LIN {X 0,Y 249.016,Z 307.091,A -85,B 0,C 180,E1 -18932.424,E2 -18932.424} C_VEL
LIN {X 0,Y 249.002,Z 307.055,A -85,B 0,C 180,E1 -18936.346,E2 -18936.346} C_VEL
LIN {X 0,Y 248.968,Z 307.097,A -85,B 0,C 180,E1 -18940.481,E2 -18940.481} C_VEL
LIN {X 0,Y 248.963,Z 307.068,A -85,B 0,C 180,E1 -18944.884,E2 -18944.884} C_VEL
LIN {X 0,Y 248.997,Z 307.08,A -85,B 0,C 180,E1 -18947.359,E2 -18947.359} C_VEL
LIN {X 0,Y 249.012,Z 307.077,A -85,B 0,C 180,E1 -18951.617,E2 -18951.617} C_VEL
LIN {X 0,Y 249.03,Z 307.09,A -85,B 0,C 180,E1 -18955.637,E2 -18955.637} C_VEL
LIN {X 0,Y 249.027,Z 307.069,A -85,B 0,C 180,E1 -18959.47,E2 -18959.47} C_VEL
LIN {X 0,Y 249.054,Z 307.084,A -85,B 0,C 180,E1 -18963.16,E2 -18963.16} C_VEL
LIN {X 0,Y 249.047,Z 307.086,A -85,B 0,C 180,E1 -18966.729,E2 -18966.729} C_VEL
LIN {X 0,Y 249.093,Z 307.073,A -85,B 0,C 180,E1 -18970.21,E2 -18970.21} C_VEL
LIN {X 0,Y 249.188,Z 307.062,A -85,B 0,C 180,E1 -18973.508,E2 -18973.508} C_VEL
LIN {X 0,Y 250.131,Z 309.782,A -85,B 0,C 180,E1 -18973.806,E2 -18973.806} C_VEL
LIN {X 0,Y 252.115,Z 312.374,A -85,B 0,C 180,E1 -18974.302,E2 -18974.302} C_VEL
LIN {X 0,Y 254.328,Z 315.703,A -85,B 0,C 180,E1 -18974.862,E2 -18974.862} C_VEL
LIN {X 0,Y 266.802,Z 335.726,A -85,B 0,C 180,E1 -18977.834,E2 -18977.834} C_VEL
LIN {X 0,Y 270.887,Z 343.151,A -85,B 0,C 180,E1 -18978.761,E2 -18978.761} C_VEL
LIN {X 0,Y 279.656,Z 361.75,A -85,B 0,C 180,E1 -18980.732,E2 -18980.732} C_VEL
LIN {X 0,Y 281.163,Z 365.318,A -85,B 0,C 180,E1 -18981.068,E2 -18981.068} C_VEL
LIN {X 0,Y 277.951,Z 432.372,A -85,B 0,C 180,E1 -18982.814,E2 -18982.814} C_VEL
LIN {X 0,Y 276.086,Z 467.971,A -85,B 0,C 180,E1 -18983.791,E2 -18983.791} C_VEL
LIN {X 0,Y 274.618,Z 483.549,A -85,B 0,C 180,E1 -18984.492,E2 -18984.492} C_VEL
LIN {X 0,Y 272.87,Z 497.522,A -85,B 0,C 180,E1 -18985.383,E2 -18985.383} C_VEL
LIN {X 0,Y 270.76,Z 510.63,A -85,B 0,C 180,E1 -18986.465,E2 -18986.465} C_VEL
LIN {X 0,Y 268.162,Z 524.603,A -85,B 0,C 180,E1 -18987.934,E2 -18987.934} C_VEL
LIN {X 0,Y 265.302,Z 537.524,A -85,B 0,C 180,E1 -18989.62,E2 -18989.62} C_VEL
LIN {X 0,Y 262.375,Z 549.476,A -85,B 0,C 180,E1 -18991.534,E2 -18991.534} C_VEL
LIN {X 0,Y 259.677,Z 559.615,A -85,B 0,C 180,E1 -18993.49,E2 -18993.49} C_VEL
LIN {X 0,Y 256.942,Z 569.913,A -85,B 0,C 180,E1 -18995.887,E2 -18995.887} C_VEL
LIN {X 0,Y 254.456,Z 578.684,A -85,B 0,C 180,E1 -18998.337,E2 -18998.337} C_VEL
LIN {X 0,Y 251.975,Z 587.261,A -85,B 0,C 180,E1 -19001.258,E2 -19001.258} C_VEL
LIN {X 0,Y 250.349,Z 593.389,A -85,B 0,C 180,E1 -19003.804,E2 -19003.804} C_VEL
LIN {X 0,Y 249.079,Z 598.519,A -85,B 0,C 180,E1 -19006.407,E2 -19006.407} C_VEL
LIN {X 0,Y 247.86,Z 603.923,A -85,B 0,C 180,E1 -19009.891,E2 -19009.891} C_VEL
LIN {X 0,Y 247.414,Z 606.081,A -85,B 0,C 180,E1 -19011.67,E2 -19011.67} C_VEL
LIN {X 0,Y 246.878,Z 608.676,A -85,B 0,C 180,E1 -19014.371,E2 -19014.371} C_VEL
LIN {X 0,Y 246.513,Z 610.789,A -85,B 0,C 180,E1 -19017.904,E2 -19017.904} C_VEL
LIN {X 0,Y 246.503,Z 611.519,A -85,B 0,C 180,E1 -19021.211,E2 -19021.211} C_VEL
LIN {X 0,Y 246.752,Z 611.025,A -85,B 0,C 180,E1 -19024.724,E2 -19024.724} C_VEL
LIN {X 0,Y 247.204,Z 609.866,A -85,B 0,C 180,E1 -19027.252,E2 -19027.252} C_VEL
LIN {X 0,Y 248.185,Z 607.218,A -85,B 0,C 180,E1 -19030.638,E2 -19030.638} C_VEL
LIN {X 0,Y 249.435,Z 603.684,A -85,B 0,C 180,E1 -19033.669,E2 -19033.669} C_VEL
LIN {X 0,Y 251.153,Z 599.042,A -85,B 0,C 180,E1 -19036.68,E2 -19036.68} C_VEL
LIN {X 0,Y 253.766,Z 592.279,A -85,B 0,C 180,E1 -19040.061,E2 -19040.061} C_VEL
LIN {X 0,Y 256.692,Z 584.864,A -85,B 0,C 180,E1 -19042.966,E2 -19042.966} C_VEL
LIN {X 0,Y 260.213,Z 575.633,A -85,B 0,C 180,E1 -19045.871,E2 -19045.871} C_VEL
LIN {X 0,Y 263.965,Z 565.524,A -85,B 0,C 180,E1 -19048.426,E2 -19048.426} C_VEL
LIN {X 0,Y 267.881,Z 554.319,A -85,B 0,C 180,E1 -19050.727,E2 -19050.727} C_VEL
LIN {X 0,Y 271.724,Z 542.18,A -85,B 0,C 180,E1 -19052.754,E2 -19052.754} C_VEL
LIN {X 0,Y 275.239,Z 529.729,A -85,B 0,C 180,E1 -19054.442,E2 -19054.442} C_VEL
LIN {X 0,Y 278.7,Z 515.562,A -85,B 0,C 180,E1 -19055.979,E2 -19055.979} C_VEL
LIN {X 0,Y 281.492,Z 501.777,A -85,B 0,C 180,E1 -19057.154,E2 -19057.154} C_VEL
LIN {X 0,Y 283.979,Z 486.513,A -85,B 0,C 180,E1 -19058.136,E2 -19058.136} C_VEL
LIN {X 0,Y 285.813,Z 471.219,A -85,B 0,C 180,E1 -19058.83,E2 -19058.83} C_VEL
LIN {X 0,Y 287.248,Z 451.285,A -85,B 0,C 180,E1 -19059.413,E2 -19059.413} C_VEL
LIN {X 0,Y 292.022,Z 372.427,A -85,B 0,C 180,E1 -19061.462,E2 -19061.462} C_VEL
LIN {X 0,Y 286.413,Z 360.627,A -85,B 0,C 180,E1 -19063.188,E2 -19063.188} C_VEL
LIN {X 0,Y 281.374,Z 351.253,A -85,B 0,C 180,E1 -19064.835,E2 -19064.835} C_VEL
LIN {X 0,Y 279.129,Z 347.273,A -85,B 0,C 180,E1 -19065.603,E2 -19065.603} C_VEL
LIN {X 0,Y 277.373,Z 345.191,A -85,B 0,C 180,E1 -19066.185,E2 -19066.185} C_VEL
LIN {X 0,Y 273.701,Z 343.752,A -85,B 0,C 180,E1 -19067.314,E2 -19067.314} C_VEL
LIN {X 0,Y 270.012,Z 342.607,A -85,B 0,C 180,E1 -19068.512,E2 -19068.512} C_VEL
LIN {X 0,Y 268.191,Z 340.919,A -85,B 0,C 180,E1 -19069.192,E2 -19069.192} C_VEL
LIN {X 0,Y 265.708,Z 337.548,A -85,B 0,C 180,E1 -19070.231,E2 -19070.231} C_VEL
LIN {X 0,Y 263.205,Z 334.014,A -85,B 0,C 180,E1 -19071.359,E2 -19071.359} C_VEL
LIN {X 0,Y 260.47,Z 330.142,A -85,B 0,C 180,E1 -19072.681,E2 -19072.681} C_VEL
LIN {X 0,Y 257.242,Z 326.198,A -85,B 0,C 180,E1 -19074.319,E2 -19074.319} C_VEL
LIN {X 0,Y 256.502,Z 324.959,A -85,B 0,C 180,E1 -19074.746,E2 -19074.746} C_VEL
LIN {X 0,Y 253.726,Z 322.405,A -85,B 0,C 180,E1 -19076.318,E2 -19076.318} C_VEL
LIN {X 0,Y 252.065,Z 319.429,A -85,B 0,C 180,E1 -19077.453,E2 -19077.453} C_VEL
LIN {X 0,Y 249.568,Z 317.316,A -85,B 0,C 180,E1 -19079.095,E2 -19079.095} C_VEL
LIN {X 0,Y 248.14,Z 314.667,A -85,B 0,C 180,E1 -19080.307,E2 -19080.307} C_VEL
LIN {X 0,Y 247.833,Z 313.854,A -85,B 0,C 180,E1 -19080.612,E2 -19080.612} C_VEL
LIN {X 0,Y 244.45,Z 312.125,A -85,B 0,C 180,E1 -19083.505,E2 -19083.505} C_VEL
LIN {X 0,Y 242.871,Z 310.007,A -85,B 0,C 180,E1 -19085.399,E2 -19085.399} C_VEL
LIN {X 0,Y 242.386,Z 308.16,A -85,B 0,C 180,E1 -19086.297,E2 -19086.297} C_VEL
LIN {X 0,Y 242.399,Z 307.915,A -85,B 0,C 180,E1 -19086.662,E2 -19086.662} C_VEL
LIN {X 0,Y 242.255,Z 307.93,A -85,B 0,C 180,E1 -19090.027,E2 -19090.027} C_VEL
LIN {X 0,Y 242.116,Z 307.948,A -85,B 0,C 180,E1 -19095.147,E2 -19095.147} C_VEL
LIN {X 0,Y 242.026,Z 307.964,A -85,B 0,C 180,E1 -19098.63,E2 -19098.63} C_VEL
LIN {X 0,Y 241.976,Z 308.133,A -85,B 0,C 180,E1 -19102.186,E2 -19102.186} C_VEL
LIN {X 0,Y 242.156,Z 308.978,A -85,B 0,C 180,E1 -19103.182,E2 -19103.182} C_VEL
LIN {X 0,Y 243.449,Z 311.446,A -85,B 0,C 180,E1 -19105.09,E2 -19105.09} C_VEL
LIN {X 0,Y 246.087,Z 314.023,A -85,B 0,C 180,E1 -19107.712,E2 -19107.712} C_VEL
LIN {X 0,Y 248.877,Z 317.269,A -85,B 0,C 180,E1 -19110.084,E2 -19110.084} C_VEL
LIN {X 0,Y 252.841,Z 322.416,A -85,B 0,C 180,E1 -19112.839,E2 -19112.839} C_VEL
LIN {X 0,Y 254.527,Z 324.821,A -85,B 0,C 180,E1 -19113.907,E2 -19113.907} C_VEL
LIN {X 0,Y 258.657,Z 330.491,A -85,B 0,C 180,E1 -19116.21,E2 -19116.21} C_VEL
LIN {X 0,Y 262.995,Z 337.089,A -85,B 0,C 180,E1 -19118.372,E2 -19118.372} C_VEL
LIN {X 0,Y 266.544,Z 342.557,A -85,B 0,C 180,E1 -19119.966,E2 -19119.966} C_VEL
LIN {X 0,Y 271.658,Z 351.022,A -85,B 0,C 180,E1 -19122.06,E2 -19122.06} C_VEL
LIN {X 0,Y 277.723,Z 362.338,A -85,B 0,C 180,E1 -19124.337,E2 -19124.337} C_VEL
LIN {X 0,Y 283.163,Z 373.979,A -85,B 0,C 180,E1 -19126.225,E2 -19126.225} C_VEL
LIN {X 0,Y 286.725,Z 382.655,A -85,B 0,C 180,E1 -19127.414,E2 -19127.414} C_VEL
LIN {X 0,Y 281.543,Z 465.569,A -85,B 0,C 180,E1 -19129.593,E2 -19129.593} C_VEL
LIN {X 0,Y 280.06,Z 483.965,A -85,B 0,C 180,E1 -19130.158,E2 -19130.158} C_VEL
LIN {X 0,Y 277.977,Z 499.11,A -85,B 0,C 180,E1 -19130.857,E2 -19130.857} C_VEL
LIN {X 0,Y 275.049,Z 514.438,A -85,B 0,C 180,E1 -19131.829,E2 -19131.829} C_VEL
LIN {X 0,Y 272.261,Z 526.889,A -85,B 0,C 180,E1 -19132.889,E2 -19132.889} C_VEL
LIN {X 0,Y 268.805,Z 540.094,A -85,B 0,C 180,E1 -19134.288,E2 -19134.288} C_VEL
LIN {X 0,Y 265.099,Z 552.623,A -85,B 0,C 180,E1 -19135.943,E2 -19135.943} C_VEL
LIN {X 0,Y 261.071,Z 564.628,A -85,B 0,C 180,E1 -19137.883,E2 -19137.883} C_VEL
LIN {X 0,Y 257.052,Z 575.653,A -85,B 0,C 180,E1 -19140.07,E2 -19140.07} C_VEL
LIN {X 0,Y 253.546,Z 585.071,A -85,B 0,C 180,E1 -19142.366,E2 -19142.366} C_VEL
LIN {X 0,Y 250.098,Z 594.176,A -85,B 0,C 180,E1 -19145.071,E2 -19145.071} C_VEL
LIN {X 0,Y 246.918,Z 601.891,A -85,B 0,C 180,E1 -19147.845,E2 -19147.845} C_VEL
LIN {X 0,Y 244.448,Z 608.314,A -85,B 0,C 180,E1 -19150.694,E2 -19150.694} C_VEL
LIN {X 0,Y 242.358,Z 614.253,A -85,B 0,C 180,E1 -19154.01,E2 -19154.01} C_VEL
LIN {X 0,Y 241.239,Z 617.803,A -85,B 0,C 180,E1 -19156.524,E2 -19156.524} C_VEL
LIN {X 0,Y 240.243,Z 621.431,A -85,B 0,C 180,E1 -19159.892,E2 -19159.892} C_VEL
LIN {X 0,Y 239.787,Z 623.867,A -85,B 0,C 180,E1 -19163.268,E2 -19163.268} C_VEL
LIN {X 0,Y 239.735,Z 625.146,A -85,B 0,C 180,E1 -19166.639,E2 -19166.639} C_VEL
LIN {X 0,Y 239.917,Z 625.227,A -85,B 0,C 180,E1 -19170.001,E2 -19170.001} C_VEL
LIN {X 0,Y 239.763,Z 624.101,A -85,B 0,C 180,E1 -19173.361,E2 -19173.361} C_VEL
LIN {X 0,Y 239.797,Z 621.778,A -85,B 0,C 180,E1 -19176.733,E2 -19176.733} C_VEL
LIN {X 0,Y 240.236,Z 618.206,A -85,B 0,C 180,E1 -19180.11,E2 -19180.11} C_VEL
LIN {X 0,Y 241.096,Z 613.285,A -85,B 0,C 180,E1 -19183.486,E2 -19183.486} C_VEL
LIN {X 0,Y 242.47,Z 606.876,A -85,B 0,C 180,E1 -19186.849,E2 -19186.849} C_VEL
LIN {X 0,Y 244.354,Z 599.957,A -85,B 0,C 180,E1 -19189.752,E2 -19189.752} C_VEL
LIN {X 0,Y 246.748,Z 591.573,A -85,B 0,C 180,E1 -19192.614,E2 -19192.614} C_VEL
LIN {X 0,Y 249.609,Z 581.609,A -85,B 0,C 180,E1 -19195.387,E2 -19195.387} C_VEL
LIN {X 0,Y 252.526,Z 571.082,A -85,B 0,C 180,E1 -19197.786,E2 -19197.786} C_VEL
LIN {X 0,Y 255.946,Z 558.736,A -85,B 0,C 180,E1 -19200.075,E2 -19200.075} C_VEL
LIN {X 0,Y 259.013,Z 546.324,A -85,B 0,C 180,E1 -19201.945,E2 -19201.945} C_VEL
LIN {X 0,Y 261.9,Z 533.658,A -85,B 0,C 180,E1 -19203.485,E2 -19203.485} C_VEL
LIN {X 0,Y 264.741,Z 518.918,A -85,B 0,C 180,E1 -19204.918,E2 -19204.918} C_VEL
LIN {X 0,Y 267.239,Z 503.525,A -85,B 0,C 180,E1 -19206.046,E2 -19206.046} C_VEL
LIN {X 0,Y 269.11,Z 488.092,A -85,B 0,C 180,E1 -19206.859,E2 -19206.859} C_VEL
LIN {X 0,Y 270.398,Z 471.788,A -85,B 0,C 180,E1 -19207.412,E2 -19207.412} C_VEL
LIN {X 0,Y 275.166,Z 376.753,A -85,B 0,C 180,E1 -19209.93,E2 -19209.93} C_VEL
LIN {X 0,Y 266.648,Z 356.753,A -85,B 0,C 180,E1 -19211.945,E2 -19211.945} C_VEL
LIN {X 0,Y 259.613,Z 342.174,A -85,B 0,C 180,E1 -19213.669,E2 -19213.669} C_VEL
LIN {X 0,Y 251.353,Z 326.644,A -85,B 0,C 180,E1 -19215.789,E2 -19215.789} C_VEL
LIN {X 0,Y 244.925,Z 315.683,A -85,B 0,C 180,E1 -19217.526,E2 -19217.526} C_VEL
LIN {X 0,Y 243.366,Z 312.658,A -85,B 0,C 180,E1 -19218.029,E2 -19218.029} C_VEL
LIN {X 0,Y 241.941,Z 307.964,A -85,B 0,C 180,E1 -19220.139,E2 -19220.139} C_VEL
LIN {X 0,Y 241.982,Z 307.956,A -85,B 0,C 180,E1 -19224.411,E2 -19224.411} C_VEL
LIN {X 0,Y 241.951,Z 307.972,A -85,B 0,C 180,E1 -19228.474,E2 -19228.474} C_VEL
LIN {X 0,Y 241.953,Z 307.967,A -85,B 0,C 180,E1 -19232.303,E2 -19232.303} C_VEL
LIN {X 0,Y 241.958,Z 307.969,A -85,B 0,C 180,E1 -19236.003,E2 -19236.003} C_VEL
LIN {X 0,Y 241.986,Z 307.968,A -85,B 0,C 180,E1 -19239.601,E2 -19239.601} C_VEL
LIN {X 0,Y 242.114,Z 307.955,A -85,B 0,C 180,E1 -19243.316,E2 -19243.316} C_VEL
LIN {X 0,Y 242.159,Z 307.905,A -85,B 0,C 180,E1 -19248.276,E2 -19248.276} C_VEL
LIN {X 0,Y 242.356,Z 307.921,A -85,B 0,C 180,E1 -19251.661,E2 -19251.661} C_VEL
LIN {X 0,Y 242.387,Z 307.912,A -85,B 0,C 180,E1 -19253.337,E2 -19253.337} C_VEL
LIN {X 0,Y 242.603,Z 307.858,A -85,B 0,C 180,E1 -19258.337,E2 -19258.337} C_VEL
LIN {X 0,Y 242.612,Z 307.89,A -85,B 0,C 180,E1 -19261.657,E2 -19261.657} C_VEL
LIN {X 0,Y 242.38,Z 307.87,A -85,B 0,C 180,E1 -19266.657,E2 -19266.657} C_VEL
LIN {X 0,Y 242.257,Z 307.924,A -85,B 0,C 180,E1 -19270.021,E2 -19270.021} C_VEL
LIN {X 0,Y 242.128,Z 307.917,A -85,B 0,C 180,E1 -19275.14,E2 -19275.14} C_VEL
LIN {X 0,Y 242.039,Z 307.926,A -85,B 0,C 180,E1 -19278.624,E2 -19278.624} C_VEL
LIN {X 0,Y 241.981,Z 307.967,A -85,B 0,C 180,E1 -19282.18,E2 -19282.18} C_VEL
LIN {X 0,Y 241.978,Z 307.931,A -85,B 0,C 180,E1 -19285.824,E2 -19285.824} C_VEL
LIN {X 0,Y 241.953,Z 307.951,A -85,B 0,C 180,E1 -19289.587,E2 -19289.587} C_VEL
LIN {X 0,Y 241.969,Z 307.962,A -85,B 0,C 180,E1 -19293.49,E2 -19293.49} C_VEL
LIN {X 0,Y 241.972,Z 307.933,A -85,B 0,C 180,E1 -19297.581,E2 -19297.581} C_VEL
LIN {X 0,Y 241.897,Z 307.978,A -85,B 0,C 180,E1 -19301.926,E2 -19301.926} C_VEL
LIN {X 0,Y 241.911,Z 307.952,A -85,B 0,C 180,E1 -19306.572,E2 -19306.572} C_VEL
LIN {X 0,Y 241.944,Z 307.973,A -85,B 0,C 180,E1 -19310.279,E2 -19310.279} C_VEL
LIN {X 0,Y 241.966,Z 307.955,A -85,B 0,C 180,E1 -19314.486,E2 -19314.486} C_VEL
LIN {X 0,Y 241.954,Z 307.955,A -85,B 0,C 180,E1 -19318.477,E2 -19318.477} C_VEL
LIN {X 0,Y 241.987,Z 307.967,A -85,B 0,C 180,E1 -19322.31,E2 -19322.31} C_VEL
LIN {X 0,Y 242.027,Z 307.952,A -85,B 0,C 180,E1 -19326.013,E2 -19326.013} C_VEL
LIN {X 0,Y 242.02,Z 307.951,A -85,B 0,C 180,E1 -19329.606,E2 -19329.606} C_VEL
LIN {X 0,Y 242.078,Z 307.956,A -85,B 0,C 180,E1 -19332.053,E2 -19332.053} C_VEL
LIN {X 0,Y 243.143,Z 310.845,A -85,B 0,C 180,E1 -19332.418,E2 -19332.418} C_VEL
LIN {X 0,Y 245.158,Z 313.379,A -85,B 0,C 180,E1 -19332.948,E2 -19332.948} C_VEL
LIN {X 0,Y 247.321,Z 316.579,A -85,B 0,C 180,E1 -19333.523,E2 -19333.523} C_VEL
LIN {X 0,Y 259.586,Z 335.968,A -85,B 0,C 180,E1 -19336.608,E2 -19336.608} C_VEL
LIN {X 0,Y 265.566,Z 346.45,A -85,B 0,C 180,E1 -19338.019,E2 -19338.019} C_VEL
LIN {X 0,Y 274.158,Z 364.708,A -85,B 0,C 180,E1 -19340.015,E2 -19340.015} C_VEL
LIN {X 0,Y 275.294,Z 367.332,A -85,B 0,C 180,E1 -19340.276,E2 -19340.276} C_VEL
LIN {X 0,Y 272.005,Z 432.87,A -85,B 0,C 180,E1 -19342.009,E2 -19342.009} C_VEL
LIN {X 0,Y 270.137,Z 467.831,A -85,B 0,C 180,E1 -19342.984,E2 -19342.984} C_VEL
LIN {X 0,Y 268.633,Z 483.311,A -85,B 0,C 180,E1 -19343.683,E2 -19343.683} C_VEL
LIN {X 0,Y 266.766,Z 497.727,A -85,B 0,C 180,E1 -19344.614,E2 -19344.614} C_VEL
LIN {X 0,Y 264.417,Z 511.816,A -85,B 0,C 180,E1 -19345.808,E2 -19345.808} C_VEL
LIN {X 0,Y 261.826,Z 525.241,A -85,B 0,C 180,E1 -19347.264,E2 -19347.264} C_VEL
LIN {X 0,Y 258.779,Z 538.408,A -85,B 0,C 180,E1 -19349.027,E2 -19349.027} C_VEL
LIN {X 0,Y 255.508,Z 551.324,A -85,B 0,C 180,E1 -19351.181,E2 -19351.181} C_VEL
LIN {X 0,Y 252.247,Z 563.048,A -85,B 0,C 180,E1 -19353.593,E2 -19353.593} C_VEL
LIN {X 0,Y 249.474,Z 572.876,A -85,B 0,C 180,E1 -19356.063,E2 -19356.063} C_VEL
LIN {X 0,Y 246.611,Z 582.487,A -85,B 0,C 180,E1 -19359.017,E2 -19359.017} C_VEL
LIN {X 0,Y 244.296,Z 590.398,A -85,B 0,C 180,E1 -19362.025,E2 -19362.025} C_VEL
LIN {X 0,Y 242.557,Z 596.906,A -85,B 0,C 180,E1 -19365.115,E2 -19365.115} C_VEL
LIN {X 0,Y 241.081,Z 602.801,A -85,B 0,C 180,E1 -19368.702,E2 -19368.702} C_VEL
LIN {X 0,Y 240.522,Z 605.453,A -85,B 0,C 180,E1 -19370.777,E2 -19370.777} C_VEL
LIN {X 0,Y 239.806,Z 608.805,A -85,B 0,C 180,E1 -19374.222,E2 -19374.222} C_VEL
LIN {X 0,Y 239.417,Z 611.011,A -85,B 0,C 180,E1 -19378.012,E2 -19378.012} C_VEL
LIN {X 0,Y 239.425,Z 611.752,A -85,B 0,C 180,E1 -19381.659,E2 -19381.659} C_VEL
LIN {X 0,Y 239.69,Z 611.275,A -85,B 0,C 180,E1 -19384.822,E2 -19384.822} C_VEL
LIN {X 0,Y 240.238,Z 609.872,A -85,B 0,C 180,E1 -19387.902,E2 -19387.902} C_VEL
LIN {X 0,Y 241.124,Z 607.734,A -85,B 0,C 180,E1 -19390.733,E2 -19390.733} C_VEL
LIN {X 0,Y 242.526,Z 604.064,A -85,B 0,C 180,E1 -19394.063,E2 -19394.063} C_VEL
LIN {X 0,Y 244.357,Z 599.457,A -85,B 0,C 180,E1 -19397.169,E2 -19397.169} C_VEL
LIN {X 0,Y 246.769,Z 593.58,A -85,B 0,C 180,E1 -19400.258,E2 -19400.258} C_VEL
LIN {X 0,Y 249.584,Z 586.808,A -85,B 0,C 180,E1 -19403.103,E2 -19403.103} C_VEL
LIN {X 0,Y 252.832,Z 578.933,A -85,B 0,C 180,E1 -19405.785,E2 -19405.785} C_VEL
LIN {X 0,Y 256.291,Z 570.214,A -85,B 0,C 180,E1 -19408.217,E2 -19408.217} C_VEL
LIN {X 0,Y 260.105,Z 560.007,A -85,B 0,C 180,E1 -19410.566,E2 -19410.566} C_VEL
LIN {X 0,Y 263.927,Z 549.071,A -85,B 0,C 180,E1 -19412.622,E2 -19412.622} C_VEL
LIN {X 0,Y 267.723,Z 537.069,A -85,B 0,C 180,E1 -19414.469,E2 -19414.469} C_VEL
LIN {X 0,Y 271.14,Z 524.776,A -85,B 0,C 180,E1 -19416.016,E2 -19416.016} C_VEL
LIN {X 0,Y 274.554,Z 510.705,A -85,B 0,C 180,E1 -19417.423,E2 -19417.423} C_VEL
LIN {X 0,Y 277.311,Z 496.463,A -85,B 0,C 180,E1 -19418.545,E2 -19418.545} C_VEL
LIN {X 0,Y 279.606,Z 481.581,A -85,B 0,C 180,E1 -19419.41,E2 -19419.41} C_VEL
LIN {X 0,Y 281.278,Z 466.673,A -85,B 0,C 180,E1 -19420.004,E2 -19420.004} C_VEL
LIN {X 0,Y 287.094,Z 375.056,A -85,B 0,C 180,E1 -19422.438,E2 -19422.438} C_VEL
LIN {X 0,Y 281.49,Z 363.189,A -85,B 0,C 180,E1 -19424.281,E2 -19424.281} C_VEL
LIN {X 0,Y 275.852,Z 352.738,A -85,B 0,C 180,E1 -19426.255,E2 -19426.255} C_VEL
LIN {X 0,Y 272.39,Z 346.926,A -85,B 0,C 180,E1 -19427.55,E2 -19427.55} C_VEL
LIN {X 0,Y 268.191,Z 340.919,A -85,B 0,C 180,E1 -19429.192,E2 -19429.192} C_VEL
LIN {X 0,Y 266.423,Z 339.37,A -85,B 0,C 180,E1 -19429.883,E2 -19429.883} C_VEL
LIN {X 0,Y 259.762,Z 338.223,A -85,B 0,C 180,E1 -19432.456,E2 -19432.456} C_VEL
LIN {X 0,Y 258.249,Z 336.615,A -85,B 0,C 180,E1 -19433.186,E2 -19433.186} C_VEL
LIN {X 0,Y 254.764,Z 331.965,A -85,B 0,C 180,E1 -19435.07,E2 -19435.07} C_VEL
LIN {X 0,Y 253,Z 330.233,A -85,B 0,C 180,E1 -19436.081,E2 -19436.081} C_VEL
LIN {X 0,Y 250.763,Z 327.162,A -85,B 0,C 180,E1 -19437.535,E2 -19437.535} C_VEL
LIN {X 0,Y 250.101,Z 326.02,A -85,B 0,C 180,E1 -19438.009,E2 -19438.009} C_VEL
LIN {X 0,Y 247.455,Z 323.32,A -85,B 0,C 180,E1 -19439.901,E2 -19439.901} C_VEL
LIN {X 0,Y 246.027,Z 320.612,A -85,B 0,C 180,E1 -19441.22,E2 -19441.22} C_VEL
LIN {X 0,Y 242.806,Z 318.7,A -85,B 0,C 180,E1 -19444.152,E2 -19444.152} C_VEL
LIN {X 0,Y 241.415,Z 316.36,A -85,B 0,C 180,E1 -19446.06,E2 -19446.06} C_VEL
LIN {X 0,Y 240.961,Z 314.87,A -85,B 0,C 180,E1 -19446.914,E2 -19446.914} C_VEL
LIN {X 0,Y 238.232,Z 313.888,A -85,B 0,C 180,E1 -19453.654,E2 -19453.654} C_VEL
LIN {X 0,Y 238.876,Z 314.332,A -85,B 0,C 180,E1 -19458.885,E2 -19458.885} C_VEL
LIN {X 0,Y 240.472,Z 315.068,A -85,B 0,C 180,E1 -19462.064,E2 -19462.064} C_VEL
LIN {X 0,Y 240.98,Z 316.088,A -85,B 0,C 180,E1 -19462.961,E2 -19462.961} C_VEL
LIN {X 0,Y 242.653,Z 318.901,A -85,B 0,C 180,E1 -19465.349,E2 -19465.349} C_VEL
LIN {X 0,Y 244.671,Z 320.82,A -85,B 0,C 180,E1 -19467.363,E2 -19467.363} C_VEL
LIN {X 0,Y 247.396,Z 324.08,A -85,B 0,C 180,E1 -19469.762,E2 -19469.762} C_VEL
LIN {X 0,Y 250.326,Z 328.216,A -85,B 0,C 180,E1 -19471.929,E2 -19471.929} C_VEL
LIN {X 0,Y 251.962,Z 330.295,A -85,B 0,C 180,E1 -19473.001,E2 -19473.001} C_VEL
LIN {X 0,Y 256.324,Z 336.686,A -85,B 0,C 180,E1 -19475.611,E2 -19475.611} C_VEL
LIN {X 0,Y 260.397,Z 343.002,A -85,B 0,C 180,E1 -19477.724,E2 -19477.724} C_VEL
LIN {X 0,Y 263.994,Z 348.761,A -85,B 0,C 180,E1 -19479.422,E2 -19479.422} C_VEL
LIN {X 0,Y 268.962,Z 357.338,A -85,B 0,C 180,E1 -19481.548,E2 -19481.548} C_VEL
LIN {X 0,Y 274.617,Z 368.304,A -85,B 0,C 180,E1 -19483.765,E2 -19483.765} C_VEL
LIN {X 0,Y 279.332,Z 378.777,A -85,B 0,C 180,E1 -19485.486,E2 -19485.486} C_VEL
LIN {X 0,Y 281.952,Z 385.263,A -85,B 0,C 180,E1 -19486.413,E2 -19486.413} C_VEL
LIN {X 0,Y 275.698,Z 478.622,A -85,B 0,C 180,E1 -19488.915,E2 -19488.915} C_VEL
LIN {X 0,Y 273.701,Z 494.637,A -85,B 0,C 180,E1 -19489.584,E2 -19489.584} C_VEL
LIN {X 0,Y 271.032,Z 509.37,A -85,B 0,C 180,E1 -19490.439,E2 -19490.439} C_VEL
LIN {X 0,Y 267.996,Z 522.795,A -85,B 0,C 180,E1 -19491.479,E2 -19491.479} C_VEL
LIN {X 0,Y 264.329,Z 536.894,A -85,B 0,C 180,E1 -19492.908,E2 -19492.908} C_VEL
LIN {X 0,Y 260.428,Z 549.686,A -85,B 0,C 180,E1 -19494.537,E2 -19494.537} C_VEL
LIN {X 0,Y 256.258,Z 562.072,A -85,B 0,C 180,E1 -19496.502,E2 -19496.502} C_VEL
LIN {X 0,Y 252.28,Z 572.561,A -85,B 0,C 180,E1 -19498.513,E2 -19498.513} C_VEL
LIN {X 0,Y 248.435,Z 582.323,A -85,B 0,C 180,E1 -19500.793,E2 -19500.793} C_VEL
LIN {X 0,Y 244.597,Z 591.931,A -85,B 0,C 180,E1 -19503.555,E2 -19503.555} C_VEL
LIN {X 0,Y 241.139,Z 599.988,A -85,B 0,C 180,E1 -19506.377,E2 -19506.377} C_VEL
LIN {X 0,Y 238.412,Z 606.702,A -85,B 0,C 180,E1 -19509.285,E2 -19509.285} C_VEL
LIN {X 0,Y 235.937,Z 612.924,A -85,B 0,C 180,E1 -19512.671,E2 -19512.671} C_VEL
LIN {X 0,Y 234.272,Z 617.766,A -85,B 0,C 180,E1 -19516.115,E2 -19516.115} C_VEL
LIN {X 0,Y 233.191,Z 621.34,A -85,B 0,C 180,E1 -19519.583,E2 -19519.583} C_VEL
LIN {X 0,Y 232.709,Z 623.721,A -85,B 0,C 180,E1 -19523.062,E2 -19523.062} C_VEL
LIN {X 0,Y 232.644,Z 624.952,A -85,B 0,C 180,E1 -19526.537,E2 -19526.537} C_VEL
LIN {X 0,Y 232.826,Z 625.011,A -85,B 0,C 180,E1 -19530.001,E2 -19530.001} C_VEL
LIN {X 0,Y 232.669,Z 623.839,A -85,B 0,C 180,E1 -19533.464,E2 -19533.464} C_VEL
LIN {X 0,Y 232.736,Z 621.468,A -85,B 0,C 180,E1 -19536.938,E2 -19536.938} C_VEL
LIN {X 0,Y 233.177,Z 617.842,A -85,B 0,C 180,E1 -19540.419,E2 -19540.419} C_VEL
LIN {X 0,Y 234.134,Z 612.866,A -85,B 0,C 180,E1 -19543.895,E2 -19543.895} C_VEL
LIN {X 0,Y 235.593,Z 606.396,A -85,B 0,C 180,E1 -19547.356,E2 -19547.356} C_VEL
LIN {X 0,Y 237.6,Z 599.412,A -85,B 0,C 180,E1 -19550.338,E2 -19550.338} C_VEL
LIN {X 0,Y 240.152,Z 590.971,A -85,B 0,C 180,E1 -19553.271,E2 -19553.271} C_VEL
LIN {X 0,Y 242.996,Z 581.341,A -85,B 0,C 180,E1 -19556.008,E2 -19556.008} C_VEL
LIN {X 0,Y 246.184,Z 570.313,A -85,B 0,C 180,E1 -19558.566,E2 -19558.566} C_VEL
LIN {X 0,Y 249.771,Z 557.816,A -85,B 0,C 180,E1 -19560.898,E2 -19560.898} C_VEL
LIN {X 0,Y 252.951,Z 545.271,A -85,B 0,C 180,E1 -19562.805,E2 -19562.805} C_VEL
LIN {X 0,Y 256.245,Z 531.062,A -85,B 0,C 180,E1 -19564.518,E2 -19564.518} C_VEL
LIN {X 0,Y 259.042,Z 516.269,A -85,B 0,C 180,E1 -19565.923,E2 -19565.923} C_VEL
LIN {X 0,Y 261.504,Z 501.472,A -85,B 0,C 180,E1 -19566.965,E2 -19566.965} C_VEL
LIN {X 0,Y 263.317,Z 486.221,A -85,B 0,C 180,E1 -19567.749,E2 -19567.749} C_VEL
LIN {X 0,Y 264.504,Z 470.602,A -85,B 0,C 180,E1 -19568.274,E2 -19568.274} C_VEL
LIN {X 0,Y 269.295,Z 378.699,A -85,B 0,C 180,E1 -19570.75,E2 -19570.75} C_VEL
LIN {X 0,Y 260.56,Z 358.235,A -85,B 0,C 180,E1 -19572.903,E2 -19572.903} C_VEL
LIN {X 0,Y 252.589,Z 342.055,A -85,B 0,C 180,E1 -19574.944,E2 -19574.944} C_VEL
LIN {X 0,Y 245.867,Z 329.597,A -85,B 0,C 180,E1 -19576.751,E2 -19576.751} C_VEL
LIN {X 0,Y 238.626,Z 317.013,A -85,B 0,C 180,E1 -19578.813,E2 -19578.813} C_VEL
LIN {X 0,Y 235.987,Z 312.514,A -85,B 0,C 180,E1 -19579.626,E2 -19579.626} C_VEL
LIN {X 0,Y 234.929,Z 308.838,A -85,B 0,C 180,E1 -19581.353,E2 -19581.353} C_VEL
LIN {X 0,Y 234.905,Z 308.83,A -85,B 0,C 180,E1 -19585.355,E2 -19585.355} C_VEL
LIN {X 0,Y 234.955,Z 308.838,A -85,B 0,C 180,E1 -19587.421,E2 -19587.421} C_VEL
LIN {X 0,Y 234.894,Z 308.853,A -85,B 0,C 180,E1 -19591.396,E2 -19591.396} C_VEL
LIN {X 0,Y 234.901,Z 308.854,A -85,B 0,C 180,E1 -19595.234,E2 -19595.234} C_VEL
LIN {X 0,Y 234.938,Z 308.852,A -85,B 0,C 180,E1 -19598.96,E2 -19598.96} C_VEL
LIN {X 0,Y 235.056,Z 308.836,A -85,B 0,C 180,E1 -19603.091,E2 -19603.091} C_VEL
LIN {X 0,Y 235.092,Z 308.782,A -85,B 0,C 180,E1 -19607.918,E2 -19607.918} C_VEL
LIN {X 0,Y 235.295,Z 308.798,A -85,B 0,C 180,E1 -19611.408,E2 -19611.408} C_VEL
LIN {X 0,Y 235.338,Z 308.792,A -85,B 0,C 180,E1 -19613.137,E2 -19613.137} C_VEL
LIN {X 0,Y 235.562,Z 308.733,A -85,B 0,C 180,E1 -19618.288,E2 -19618.288} C_VEL
LIN {X 0,Y 235.572,Z 308.767,A -85,B 0,C 180,E1 -19621.707,E2 -19621.707} C_VEL
LIN {X 0,Y 235.331,Z 308.747,A -85,B 0,C 180,E1 -19626.858,E2 -19626.858} C_VEL
LIN {X 0,Y 235.205,Z 308.807,A -85,B 0,C 180,E1 -19630.325,E2 -19630.325} C_VEL
LIN {X 0,Y 235.073,Z 308.788,A -85,B 0,C 180,E1 -19635.606,E2 -19635.606} C_VEL
LIN {X 0,Y 234.979,Z 308.814,A -85,B 0,C 180,E1 -19639.205,E2 -19639.205} C_VEL
LIN {X 0,Y 234.917,Z 308.846,A -85,B 0,C 180,E1 -19642.884,E2 -19642.884} C_VEL
LIN {X 0,Y 234.896,Z 308.805,A -85,B 0,C 180,E1 -19646.663,E2 -19646.663} C_VEL
LIN {X 0,Y 234.885,Z 308.845,A -85,B 0,C 180,E1 -19650.57,E2 -19650.57} C_VEL
LIN {X 0,Y 234.912,Z 308.825,A -85,B 0,C 180,E1 -19654.637,E2 -19654.637} C_VEL
LIN {X 0,Y 234.902,Z 308.831,A -85,B 0,C 180,E1 -19658.933,E2 -19658.933} C_VEL
LIN {X 0,Y 234.846,Z 308.84,A -85,B 0,C 180,E1 -19663.491,E2 -19663.491} C_VEL
LIN {X 0,Y 234.864,Z 308.828,A -85,B 0,C 180,E1 -19666.509,E2 -19666.509} C_VEL
LIN {X 0,Y 234.906,Z 308.84,A -85,B 0,C 180,E1 -19671.076,E2 -19671.076} C_VEL
LIN {X 0,Y 234.912,Z 308.844,A -85,B 0,C 180,E1 -19675.359,E2 -19675.359} C_VEL
LIN {X 0,Y 234.906,Z 308.827,A -85,B 0,C 180,E1 -19679.428,E2 -19679.428} C_VEL
LIN {X 0,Y 234.98,Z 308.83,A -85,B 0,C 180,E1 -19683.792,E2 -19683.792} C_VEL
LIN {X 0,Y 234.983,Z 308.829,A -85,B 0,C 180,E1 -19688.967,E2 -19688.967} C_VEL
LIN {X 0,Y 234.972,Z 308.885,A -85,B 0,C 180,E1 -19690.507,E2 -19690.507} C_VEL
LIN {X 0,Y 236.026,Z 311.746,A -85,B 0,C 180,E1 -19690.88,E2 -19690.88} C_VEL
LIN {X 0,Y 238.141,Z 314.287,A -85,B 0,C 180,E1 -19691.473,E2 -19691.473} C_VEL
LIN {X 0,Y 240.536,Z 317.789,A -85,B 0,C 180,E1 -19692.155,E2 -19692.155} C_VEL
LIN {X 0,Y 248.885,Z 330.678,A -85,B 0,C 180,E1 -19694.41,E2 -19694.41} C_VEL
LIN {X 0,Y 259.076,Z 347.4,A -85,B 0,C 180,E1 -19696.948,E2 -19696.948} C_VEL
LIN {X 0,Y 268.888,Z 368.136,A -85,B 0,C 180,E1 -19699.328,E2 -19699.328} C_VEL
LIN {X 0,Y 269.506,Z 369.78,A -85,B 0,C 180,E1 -19699.482,E2 -19699.482} C_VEL
LIN {X 0,Y 264.27,Z 466.924,A -85,B 0,C 180,E1 -19702.118,E2 -19702.118} C_VEL
LIN {X 0,Y 262.699,Z 482.91,A -85,B 0,C 180,E1 -19702.837,E2 -19702.837} C_VEL
LIN {X 0,Y 260.726,Z 497.8,A -85,B 0,C 180,E1 -19703.81,E2 -19703.81} C_VEL
LIN {X 0,Y 258.451,Z 510.951,A -85,B 0,C 180,E1 -19704.929,E2 -19704.929} C_VEL
LIN {X 0,Y 255.701,Z 524.925,A -85,B 0,C 180,E1 -19706.454,E2 -19706.454} C_VEL
LIN {X 0,Y 252.737,Z 537.411,A -85,B 0,C 180,E1 -19708.137,E2 -19708.137} C_VEL
LIN {X 0,Y 249.489,Z 549.849,A -85,B 0,C 180,E1 -19710.201,E2 -19710.201} C_VEL
LIN {X 0,Y 246.205,Z 561.342,A -85,B 0,C 180,E1 -19712.54,E2 -19712.54} C_VEL
LIN {X 0,Y 243.393,Z 571.102,A -85,B 0,C 180,E1 -19714.969,E2 -19714.969} C_VEL
LIN {X 0,Y 240.508,Z 580.475,A -85,B 0,C 180,E1 -19717.788,E2 -19717.788} C_VEL
LIN {X 0,Y 238.113,Z 588.21,A -85,B 0,C 180,E1 -19720.629,E2 -19720.629} C_VEL
LIN {X 0,Y 236.092,Z 595.16,A -85,B 0,C 180,E1 -19723.776,E2 -19723.776} C_VEL
LIN {X 0,Y 234.718,Z 600.285,A -85,B 0,C 180,E1 -19726.647,E2 -19726.647} C_VEL
LIN {X 0,Y 233.619,Z 605.1,A -85,B 0,C 180,E1 -19730.146,E2 -19730.146} C_VEL
LIN {X 0,Y 232.873,Z 608.1,A -85,B 0,C 180,E1 -19733.099,E2 -19733.099} C_VEL
LIN {X 0,Y 232.569,Z 609.584,A -85,B 0,C 180,E1 -19735.027,E2 -19735.027} C_VEL
LIN {X 0,Y 232.27,Z 611.475,A -85,B 0,C 180,E1 -19738.954,E2 -19738.954} C_VEL
LIN {X 0,Y 232.337,Z 611.945,A -85,B 0,C 180,E1 -19742.123,E2 -19742.123} C_VEL
LIN {X 0,Y 232.656,Z 611.42,A -85,B 0,C 180,E1 -19745.359,E2 -19745.359} C_VEL
LIN {X 0,Y 233.498,Z 609.507,A -85,B 0,C 180,E1 -19749.201,E2 -19749.201} C_VEL
LIN {X 0,Y 234.655,Z 606.815,A -85,B 0,C 180,E1 -19752.364,E2 -19752.364} C_VEL
LIN {X 0,Y 236.223,Z 603.054,A -85,B 0,C 180,E1 -19755.562,E2 -19755.562} C_VEL
LIN {X 0,Y 238.32,Z 598.185,A -85,B 0,C 180,E1 -19758.709,E2 -19758.709} C_VEL
LIN {X 0,Y 241.101,Z 591.823,A -85,B 0,C 180,E1 -19761.907,E2 -19761.907} C_VEL
LIN {X 0,Y 244.406,Z 584.328,A -85,B 0,C 180,E1 -19764.897,E2 -19764.897} C_VEL
LIN {X 0,Y 248.03,Z 575.884,A -85,B 0,C 180,E1 -19767.62,E2 -19767.62} C_VEL
LIN {X 0,Y 252.053,Z 566.022,A -85,B 0,C 180,E1 -19770.207,E2 -19770.207} C_VEL
LIN {X 0,Y 256.385,Z 554.685,A -85,B 0,C 180,E1 -19772.609,E2 -19772.609} C_VEL
LIN {X 0,Y 260.627,Z 542.538,A -85,B 0,C 180,E1 -19774.688,E2 -19774.688} C_VEL
LIN {X 0,Y 264.291,Z 530.592,A -85,B 0,C 180,E1 -19776.358,E2 -19776.358} C_VEL
LIN {X 0,Y 268.092,Z 516.271,A -85,B 0,C 180,E1 -19777.96,E2 -19777.96} C_VEL
LIN {X 0,Y 271.162,Z 502.384,A -85,B 0,C 180,E1 -19779.17,E2 -19779.17} C_VEL
LIN {X 0,Y 273.851,Z 487.187,A -85,B 0,C 180,E1 -19780.169,E2 -19780.169} C_VEL
LIN {X 0,Y 275.877,Z 471.479,A -85,B 0,C 180,E1 -19780.898,E2 -19780.898} C_VEL
LIN {X 0,Y 277.575,Z 448.975,A -85,B 0,C 180,E1 -19781.559,E2 -19781.559} C_VEL
LIN {X 0,Y 282.301,Z 377.818,A -85,B 0,C 180,E1 -19783.449,E2 -19783.449} C_VEL
LIN {X 0,Y 276.87,Z 366.28,A -85,B 0,C 180,E1 -19785.337,E2 -19785.337} C_VEL
LIN {X 0,Y 270.801,Z 354.928,A -85,B 0,C 180,E1 -19787.629,E2 -19787.629} C_VEL
LIN {X 0,Y 265.717,Z 347.206,A -85,B 0,C 180,E1 -19789.689,E2 -19789.689} C_VEL
LIN {X 0,Y 260.792,Z 340.205,A -85,B 0,C 180,E1 -19791.918,E2 -19791.918} C_VEL
LIN {X 0,Y 258.249,Z 336.615,A -85,B 0,C 180,E1 -19793.186,E2 -19793.186} C_VEL
LIN {X 0,Y 256.931,Z 334.75,A -85,B 0,C 180,E1 -19793.882,E2 -19793.882} C_VEL
LIN {X 0,Y 255.43,Z 333.622,A -85,B 0,C 180,E1 -19794.645,E2 -19794.645} C_VEL
LIN {X 0,Y 252.256,Z 332.783,A -85,B 0,C 180,E1 -19796.272,E2 -19796.272} C_VEL
LIN {X 0,Y 249.166,Z 332.487,A -85,B 0,C 180,E1 -19797.997,E2 -19797.997} C_VEL
LIN {X 0,Y 247.165,Z 331.568,A -85,B 0,C 180,E1 -19799.301,E2 -19799.301} C_VEL
LIN {X 0,Y 246.592,Z 330.982,A -85,B 0,C 180,E1 -19799.729,E2 -19799.729} C_VEL
LIN {X 0,Y 244.784,Z 327.86,A -85,B 0,C 180,E1 -19801.366,E2 -19801.366} C_VEL
LIN {X 0,Y 244.478,Z 327.436,A -85,B 0,C 180,E1 -19801.65,E2 -19801.65} C_VEL
LIN {X 0,Y 241.413,Z 325.437,A -85,B 0,C 180,E1 -19804.595,E2 -19804.595} C_VEL
LIN {X 0,Y 240.083,Z 323.076,A -85,B 0,C 180,E1 -19806.542,E2 -19806.542} C_VEL
LIN {X 0,Y 239.645,Z 321.827,A -85,B 0,C 180,E1 -19807.374,E2 -19807.374} C_VEL
LIN {X 0,Y 237.246,Z 320.9,A -85,B 0,C 180,E1 -19813.711,E2 -19813.711} C_VEL
LIN {X 0,Y 237.955,Z 321.401,A -85,B 0,C 180,E1 -19819.076,E2 -19819.076} C_VEL
LIN {X 0,Y 239.374,Z 322.058,A -85,B 0,C 180,E1 -19821.9,E2 -19821.9} C_VEL
LIN {X 0,Y 241.107,Z 325.417,A -85,B 0,C 180,E1 -19824.701,E2 -19824.701} C_VEL
LIN {X 0,Y 243.329,Z 327.682,A -85,B 0,C 180,E1 -19827.073,E2 -19827.073} C_VEL
LIN {X 0,Y 245.711,Z 330.665,A -85,B 0,C 180,E1 -19829.251,E2 -19829.251} C_VEL
LIN {X 0,Y 249.148,Z 335.474,A -85,B 0,C 180,E1 -19831.874,E2 -19831.874} C_VEL
LIN {X 0,Y 254.044,Z 342.859,A -85,B 0,C 180,E1 -19835.004,E2 -19835.004} C_VEL
LIN {X 0,Y 257.704,Z 348.712,A -85,B 0,C 180,E1 -19836.997,E2 -19836.997} C_VEL
LIN {X 0,Y 261.099,Z 354.286,A -85,B 0,C 180,E1 -19838.688,E2 -19838.688} C_VEL
LIN {X 0,Y 265.776,Z 362.669,A -85,B 0,C 180,E1 -19840.804,E2 -19840.804} C_VEL
LIN {X 0,Y 271.097,Z 373.273,A -85,B 0,C 180,E1 -19842.996,E2 -19842.996} C_VEL
LIN {X 0,Y 275.444,Z 383.276,A -85,B 0,C 180,E1 -19844.684,E2 -19844.684} C_VEL
LIN {X 0,Y 277.24,Z 387.736,A -85,B 0,C 180,E1 -19845.349,E2 -19845.349} C_VEL
LIN {X 0,Y 270.98,Z 477.662,A -85,B 0,C 180,E1 -19847.789,E2 -19847.789} C_VEL
LIN {X 0,Y 268.927,Z 493.907,A -85,B 0,C 180,E1 -19848.462,E2 -19848.462} C_VEL
LIN {X 0,Y 266.177,Z 508.701,A -85,B 0,C 180,E1 -19849.322,E2 -19849.322} C_VEL
LIN {X 0,Y 263.018,Z 522.186,A -85,B 0,C 180,E1 -19850.362,E2 -19850.362} C_VEL
LIN {X 0,Y 259.186,Z 536.395,A -85,B 0,C 180,E1 -19851.802,E2 -19851.802} C_VEL
LIN {X 0,Y 255.137,Z 549.218,A -85,B 0,C 180,E1 -19853.44,E2 -19853.44} C_VEL
LIN {X 0,Y 250.784,Z 561.65,A -85,B 0,C 180,E1 -19855.426,E2 -19855.426} C_VEL
LIN {X 0,Y 246.273,Z 573.027,A -85,B 0,C 180,E1 -19857.652,E2 -19857.652} C_VEL
LIN {X 0,Y 242.245,Z 582.649,A -85,B 0,C 180,E1 -19859.971,E2 -19859.971} C_VEL
LIN {X 0,Y 238.228,Z 592.16,A -85,B 0,C 180,E1 -19862.791,E2 -19862.791} C_VEL
LIN {X 0,Y 234.62,Z 600.139,A -85,B 0,C 180,E1 -19865.678,E2 -19865.678} C_VEL
LIN {X 0,Y 231.721,Z 606.806,A -85,B 0,C 180,E1 -19868.658,E2 -19868.658} C_VEL
LIN {X 0,Y 229.097,Z 612.957,A -85,B 0,C 180,E1 -19872.137,E2 -19872.137} C_VEL
LIN {X 0,Y 227.327,Z 617.729,A -85,B 0,C 180,E1 -19875.682,E2 -19875.682} C_VEL
LIN {X 0,Y 226.156,Z 621.25,A -85,B 0,C 180,E1 -19879.255,E2 -19879.255} C_VEL
LIN {X 0,Y 225.622,Z 623.579,A -85,B 0,C 180,E1 -19882.843,E2 -19882.843} C_VEL
LIN {X 0,Y 225.541,Z 624.759,A -85,B 0,C 180,E1 -19886.428,E2 -19886.428} C_VEL
LIN {X 0,Y 225.738,Z 624.788,A -85,B 0,C 180,E1 -19890.001,E2 -19890.001} C_VEL
LIN {X 0,Y 225.578,Z 623.571,A -85,B 0,C 180,E1 -19893.573,E2 -19893.573} C_VEL
LIN {X 0,Y 225.649,Z 621.149,A -85,B 0,C 180,E1 -19897.157,E2 -19897.157} C_VEL
LIN {X 0,Y 226.143,Z 617.467,A -85,B 0,C 180,E1 -19900.747,E2 -19900.747} C_VEL
LIN {X 0,Y 227.185,Z 612.43,A -85,B 0,C 180,E1 -19904.329,E2 -19904.329} C_VEL
LIN {X 0,Y 228.784,Z 605.894,A -85,B 0,C 180,E1 -19907.89,E2 -19907.89} C_VEL
LIN {X 0,Y 230.852,Z 598.828,A -85,B 0,C 180,E1 -19910.96,E2 -19910.96} C_VEL
LIN {X 0,Y 233.576,Z 590.303,A -85,B 0,C 180,E1 -19913.966,E2 -19913.966} C_VEL
LIN {X 0,Y 236.555,Z 580.406,A -85,B 0,C 180,E1 -19916.819,E2 -19916.819} C_VEL
LIN {X 0,Y 239.884,Z 569.43,A -85,B 0,C 180,E1 -19919.389,E2 -19919.389} C_VEL
LIN {X 0,Y 243.308,Z 557.97,A -85,B 0,C 180,E1 -19921.57,E2 -19921.57} C_VEL
LIN {X 0,Y 246.586,Z 545.482,A -85,B 0,C 180,E1 -19923.519,E2 -19923.519} C_VEL
LIN {X 0,Y 249.978,Z 531.388,A -85,B 0,C 180,E1 -19925.265,E2 -19925.265} C_VEL
LIN {X 0,Y 252.86,Z 516.742,A -85,B 0,C 180,E1 -19926.696,E2 -19926.696} C_VEL
LIN {X 0,Y 255.494,Z 501.422,A -85,B 0,C 180,E1 -19927.799,E2 -19927.799} C_VEL
LIN {X 0,Y 257.367,Z 486.252,A -85,B 0,C 180,E1 -19928.594,E2 -19928.594} C_VEL
LIN {X 0,Y 258.59,Z 470.767,A -85,B 0,C 180,E1 -19929.127,E2 -19929.127} C_VEL
LIN {X 0,Y 263.453,Z 380.824,A -85,B 0,C 180,E1 -19931.593,E2 -19931.593} C_VEL
LIN {X 0,Y 255.673,Z 362.32,A -85,B 0,C 180,E1 -19933.6,E2 -19933.6} C_VEL
LIN {X 0,Y 248.364,Z 347.316,A -85,B 0,C 180,E1 -19935.533,E2 -19935.533} C_VEL
LIN {X 0,Y 241.61,Z 334.492,A -85,B 0,C 180,E1 -19937.425,E2 -19937.425} C_VEL
LIN {X 0,Y 234.33,Z 321.814,A -85,B 0,C 180,E1 -19939.563,E2 -19939.563} C_VEL
LIN {X 0,Y 230.623,Z 315.859,A -85,B 0,C 180,E1 -19940.71,E2 -19940.71} C_VEL
LIN {X 0,Y 228.646,Z 312.211,A -85,B 0,C 180,E1 -19941.403,E2 -19941.403} C_VEL
LIN {X 0,Y 227.884,Z 309.731,A -85,B 0,C 180,E1 -19942.691,E2 -19942.691} C_VEL
LIN {X 0,Y 227.88,Z 309.707,A -85,B 0,C 180,E1 -19946.377,E2 -19946.377} C_VEL
LIN {X 0,Y 227.874,Z 309.723,A -85,B 0,C 180,E1 -19950.429,E2 -19950.429} C_VEL
LIN {X 0,Y 227.868,Z 309.731,A -85,B 0,C 180,E1 -19954.416,E2 -19954.416} C_VEL
LIN {X 0,Y 227.92,Z 309.727,A -85,B 0,C 180,E1 -19958.28,E2 -19958.28} C_VEL
LIN {X 0,Y 228.018,Z 309.705,A -85,B 0,C 180,E1 -19963.892,E2 -19963.892} C_VEL
LIN {X 0,Y 228.126,Z 309.664,A -85,B 0,C 180,E1 -19969.345,E2 -19969.345} C_VEL
LIN {X 0,Y 228.29,Z 309.673,A -85,B 0,C 180,E1 -19972.924,E2 -19972.924} C_VEL
LIN {X 0,Y 228.495,Z 309.612,A -85,B 0,C 180,E1 -19978.235,E2 -19978.235} C_VEL
LIN {X 0,Y 228.53,Z 309.643,A -85,B 0,C 180,E1 -19981.759,E2 -19981.759} C_VEL
LIN {X 0,Y 228.268,Z 309.627,A -85,B 0,C 180,E1 -19987.071,E2 -19987.071} C_VEL
LIN {X 0,Y 228.136,Z 309.689,A -85,B 0,C 180,E1 -19990.648,E2 -19990.648} C_VEL
LIN {X 0,Y 228.031,Z 309.684,A -85,B 0,C 180,E1 -19994.271,E2 -19994.271} C_VEL
LIN {X 0,Y 227.931,Z 309.673,A -85,B 0,C 180,E1 -19997.956,E2 -19997.956} C_VEL
LIN {X 0,Y 227.9,Z 309.721,A -85,B 0,C 180,E1 -20002.311,E2 -20002.311} C_VEL
LIN {X 0,Y 227.862,Z 309.681,A -85,B 0,C 180,E1 -20006.562,E2 -20006.562} C_VEL
LIN {X 0,Y 227.86,Z 309.715,A -85,B 0,C 180,E1 -20010.276,E2 -20010.276} C_VEL
LIN {X 0,Y 227.866,Z 309.718,A -85,B 0,C 180,E1 -20013.718,E2 -20013.718} C_VEL
LIN {X 0,Y 227.83,Z 309.698,A -85,B 0,C 180,E1 -20018.089,E2 -20018.089} C_VEL
LIN {X 0,Y 227.776,Z 309.729,A -85,B 0,C 180,E1 -20022.745,E2 -20022.745} C_VEL
LIN {X 0,Y 227.793,Z 309.718,A -85,B 0,C 180,E1 -20027.254,E2 -20027.254} C_VEL
LIN {X 0,Y 227.828,Z 309.71,A -85,B 0,C 180,E1 -20031.906,E2 -20031.906} C_VEL
LIN {X 0,Y 227.866,Z 309.729,A -85,B 0,C 180,E1 -20036.376,E2 -20036.376} C_VEL
LIN {X 0,Y 227.889,Z 309.703,A -85,B 0,C 180,E1 -20040.433,E2 -20040.433} C_VEL
LIN {X 0,Y 227.911,Z 309.705,A -85,B 0,C 180,E1 -20044.424,E2 -20044.424} C_VEL
LIN {X 0,Y 227.941,Z 309.736,A -85,B 0,C 180,E1 -20048.858,E2 -20048.858} C_VEL
LIN {X 0,Y 228.967,Z 312.599,A -85,B 0,C 180,E1 -20049.249,E2 -20049.249} C_VEL
LIN {X 0,Y 231.12,Z 315.219,A -85,B 0,C 180,E1 -20049.893,E2 -20049.893} C_VEL
LIN {X 0,Y 233.266,Z 318.465,A -85,B 0,C 180,E1 -20050.546,E2 -20050.546} C_VEL
LIN {X 0,Y 239.79,Z 328.005,A -85,B 0,C 180,E1 -20052.434,E2 -20052.434} C_VEL
LIN {X 0,Y 251.215,Z 346.411,A -85,B 0,C 180,E1 -20055.489,E2 -20055.489} C_VEL
LIN {X 0,Y 255.927,Z 354.853,A -85,B 0,C 180,E1 -20056.674,E2 -20056.674} C_VEL
LIN {X 0,Y 263.631,Z 371.644,A -85,B 0,C 180,E1 -20058.615,E2 -20058.615} C_VEL
LIN {X 0,Y 258.396,Z 466.721,A -85,B 0,C 180,E1 -20061.248,E2 -20061.248} C_VEL
LIN {X 0,Y 256.863,Z 482.149,A -85,B 0,C 180,E1 -20061.939,E2 -20061.939} C_VEL
LIN {X 0,Y 254.707,Z 497.9,A -85,B 0,C 180,E1 -20062.973,E2 -20062.973} C_VEL
LIN {X 0,Y 252.212,Z 511.975,A -85,B 0,C 180,E1 -20064.202,E2 -20064.202} C_VEL
LIN {X 0,Y 249.359,Z 525.802,A -85,B 0,C 180,E1 -20065.757,E2 -20065.757} C_VEL
LIN {X 0,Y 246.191,Z 538.588,A -85,B 0,C 180,E1 -20067.535,E2 -20067.535} C_VEL
LIN {X 0,Y 242.616,Z 551.64,A -85,B 0,C 180,E1 -20069.792,E2 -20069.792} C_VEL
LIN {X 0,Y 239.132,Z 563.399,A -85,B 0,C 180,E1 -20072.321,E2 -20072.321} C_VEL
LIN {X 0,Y 235.885,Z 573.961,A -85,B 0,C 180,E1 -20075.127,E2 -20075.127} C_VEL
LIN {X 0,Y 233.182,Z 582.433,A -85,B 0,C 180,E1 -20077.867,E2 -20077.867} C_VEL
LIN {X 0,Y 230.446,Z 591,A -85,B 0,C 180,E1 -20081.294,E2 -20081.294} C_VEL
LIN {X 0,Y 228.736,Z 596.858,A -85,B 0,C 180,E1 -20084.228,E2 -20084.228} C_VEL
LIN {X 0,Y 227.102,Z 602.855,A -85,B 0,C 180,E1 -20088.026,E2 -20088.026} C_VEL
LIN {X 0,Y 226.188,Z 606.639,A -85,B 0,C 180,E1 -20091.239,E2 -20091.239} C_VEL
LIN {X 0,Y 225.624,Z 609.017,A -85,B 0,C 180,E1 -20093.886,E2 -20093.886} C_VEL
LIN {X 0,Y 225.212,Z 611.326,A -85,B 0,C 180,E1 -20097.909,E2 -20097.909} C_VEL
LIN {X 0,Y 225.151,Z 611.936,A -85,B 0,C 180,E1 -20099.961,E2 -20099.961} C_VEL
LIN {X 0,Y 225.272,Z 612.132,A -85,B 0,C 180,E1 -20102.619,E2 -20102.619} C_VEL
LIN {X 0,Y 225.689,Z 611.439,A -85,B 0,C 180,E1 -20106.273,E2 -20106.273} C_VEL
LIN {X 0,Y 226.366,Z 610.044,A -85,B 0,C 180,E1 -20109.094,E2 -20109.094} C_VEL
LIN {X 0,Y 227.712,Z 607.153,A -85,B 0,C 180,E1 -20112.763,E2 -20112.763} C_VEL
LIN {X 0,Y 229.379,Z 603.456,A -85,B 0,C 180,E1 -20116.053,E2 -20116.053} C_VEL
LIN {X 0,Y 231.653,Z 598.565,A -85,B 0,C 180,E1 -20119.326,E2 -20119.326} C_VEL
LIN {X 0,Y 234.89,Z 591.654,A -85,B 0,C 180,E1 -20122.886,E2 -20122.886} C_VEL
LIN {X 0,Y 238.408,Z 584.063,A -85,B 0,C 180,E1 -20125.942,E2 -20125.942} C_VEL
LIN {X 0,Y 242.787,Z 574.375,A -85,B 0,C 180,E1 -20129.055,E2 -20129.055} C_VEL
LIN {X 0,Y 247.265,Z 563.774,A -85,B 0,C 180,E1 -20131.773,E2 -20131.773} C_VEL
LIN {X 0,Y 251.845,Z 552.151,A -85,B 0,C 180,E1 -20134.15,E2 -20134.15} C_VEL
LIN {X 0,Y 256.088,Z 540.114,A -85,B 0,C 180,E1 -20136.144,E2 -20136.144} C_VEL
LIN {X 0,Y 259.823,Z 528.133,A -85,B 0,C 180,E1 -20137.751,E2 -20137.751} C_VEL
LIN {X 0,Y 263.603,Z 514.152,A -85,B 0,C 180,E1 -20139.252,E2 -20139.252} C_VEL
LIN {X 0,Y 266.615,Z 500.579,A -85,B 0,C 180,E1 -20140.4,E2 -20140.4} C_VEL
LIN {X 0,Y 269.237,Z 485.763,A -85,B 0,C 180,E1 -20141.351,E2 -20141.351} C_VEL
LIN {X 0,Y 271.205,Z 470.78,A -85,B 0,C 180,E1 -20142.024,E2 -20142.024} C_VEL
LIN {X 0,Y 273.143,Z 445.109,A -85,B 0,C 180,E1 -20142.772,E2 -20142.772} C_VEL
LIN {X 0,Y 277.596,Z 380.511,A -85,B 0,C 180,E1 -20144.507,E2 -20144.507} C_VEL
LIN {X 0,Y 272.171,Z 368.888,A -85,B 0,C 180,E1 -20146.533,E2 -20146.533} C_VEL
LIN {X 0,Y 267.092,Z 359.411,A -85,B 0,C 180,E1 -20148.563,E2 -20148.563} C_VEL
LIN {X 0,Y 261.518,Z 350.837,A -85,B 0,C 180,E1 -20150.986,E2 -20150.986} C_VEL
LIN {X 0,Y 257.721,Z 345.541,A -85,B 0,C 180,E1 -20152.826,E2 -20152.826} C_VEL
LIN {X 0,Y 255.065,Z 341.685,A -85,B 0,C 180,E1 -20154.231,E2 -20154.231} C_VEL
LIN {X 0,Y 252.065,Z 337.664,A -85,B 0,C 180,E1 -20155.984,E2 -20155.984} C_VEL
LIN {X 0,Y 249.355,Z 334.479,A -85,B 0,C 180,E1 -20157.714,E2 -20157.714} C_VEL
LIN {X 0,Y 248.162,Z 332.524,A -85,B 0,C 180,E1 -20158.583,E2 -20158.583} C_VEL
LIN {X 0,Y 246.592,Z 330.982,A -85,B 0,C 180,E1 -20159.729,E2 -20159.729} C_VEL
LIN {X 0,Y 245.443,Z 330.398,A -85,B 0,C 180,E1 -20160.597,E2 -20160.597} C_VEL
LIN {X 0,Y 243.365,Z 331.459,A -85,B 0,C 180,E1 -20162.072,E2 -20162.072} C_VEL
LIN {X 0,Y 241.407,Z 332.803,A -85,B 0,C 180,E1 -20163.584,E2 -20163.584} C_VEL
LIN {X 0,Y 240.47,Z 332.623,A -85,B 0,C 180,E1 -20164.515,E2 -20164.515} C_VEL
LIN {X 0,Y 238.856,Z 330.009,A -85,B 0,C 180,E1 -20166.868,E2 -20166.868} C_VEL
LIN {X 0,Y 238.486,Z 328.815,A -85,B 0,C 180,E1 -20167.623,E2 -20167.623} C_VEL
LIN {X 0,Y 236.264,Z 327.93,A -85,B 0,C 180,E1 -20173.769,E2 -20173.769} C_VEL
LIN {X 0,Y 236.961,Z 328.429,A -85,B 0,C 180,E1 -20179.044,E2 -20179.044} C_VEL
LIN {X 0,Y 238.279,Z 329.05,A -85,B 0,C 180,E1 -20181.736,E2 -20181.736} C_VEL
LIN {X 0,Y 239.441,Z 331.67,A -85,B 0,C 180,E1 -20183.805,E2 -20183.805} C_VEL
LIN {X 0,Y 241.998,Z 334.593,A -85,B 0,C 180,E1 -20186.789,E2 -20186.789} C_VEL
LIN {X 0,Y 243.966,Z 337.051,A -85,B 0,C 180,E1 -20188.65,E2 -20188.65} C_VEL
LIN {X 0,Y 247.382,Z 342.06,A -85,B 0,C 180,E1 -20191.418,E2 -20191.418} C_VEL
LIN {X 0,Y 251.756,Z 348.906,A -85,B 0,C 180,E1 -20194.338,E2 -20194.338} C_VEL
LIN {X 0,Y 255.841,Z 355.721,A -85,B 0,C 180,E1 -20196.673,E2 -20196.673} C_VEL
LIN {X 0,Y 258.668,Z 360.584,A -85,B 0,C 180,E1 -20198.134,E2 -20198.134} C_VEL
LIN {X 0,Y 263.048,Z 368.745,A -85,B 0,C 180,E1 -20200.211,E2 -20200.211} C_VEL
LIN {X 0,Y 267.694,Z 378.419,A -85,B 0,C 180,E1 -20202.236,E2 -20202.236} C_VEL
LIN {X 0,Y 271.684,Z 387.877,A -85,B 0,C 180,E1 -20203.871,E2 -20203.871} C_VEL
LIN {X 0,Y 272.669,Z 390.799,A -85,B 0,C 180,E1 -20204.286,E2 -20204.286} C_VEL
LIN {X 0,Y 266.261,Z 478.223,A -85,B 0,C 180,E1 -20206.666,E2 -20206.666} C_VEL
LIN {X 0,Y 264.124,Z 494.147,A -85,B 0,C 180,E1 -20207.339,E2 -20207.339} C_VEL
LIN {X 0,Y 261.165,Z 509.383,A -85,B 0,C 180,E1 -20208.241,E2 -20208.241} C_VEL
LIN {X 0,Y 257.662,Z 523.614,A -85,B 0,C 180,E1 -20209.369,E2 -20209.369} C_VEL
LIN {X 0,Y 253.703,Z 537.455,A -85,B 0,C 180,E1 -20210.82,E2 -20210.82} C_VEL
LIN {X 0,Y 249.093,Z 551.221,A -85,B 0,C 180,E1 -20212.657,E2 -20212.657} C_VEL
LIN {X 0,Y 244.997,Z 562.288,A -85,B 0,C 180,E1 -20214.488,E2 -20214.488} C_VEL
LIN {X 0,Y 240.329,Z 573.528,A -85,B 0,C 180,E1 -20216.75,E2 -20216.75} C_VEL
LIN {X 0,Y 236.128,Z 583.035,A -85,B 0,C 180,E1 -20219.11,E2 -20219.11} C_VEL
LIN {X 0,Y 231.904,Z 592.425,A -85,B 0,C 180,E1 -20221.984,E2 -20221.984} C_VEL
LIN {X 0,Y 228.148,Z 600.295,A -85,B 0,C 180,E1 -20224.942,E2 -20224.942} C_VEL
LIN {X 0,Y 225.069,Z 606.89,A -85,B 0,C 180,E1 -20227.995,E2 -20227.995} C_VEL
LIN {X 0,Y 222.269,Z 612.992,A -85,B 0,C 180,E1 -20231.568,E2 -20231.568} C_VEL
LIN {X 0,Y 220.403,Z 617.714,A -85,B 0,C 180,E1 -20235.222,E2 -20235.222} C_VEL
LIN {X 0,Y 219.14,Z 621.166,A -85,B 0,C 180,E1 -20238.907,E2 -20238.907} C_VEL
LIN {X 0,Y 218.558,Z 623.438,A -85,B 0,C 180,E1 -20242.611,E2 -20242.611} C_VEL
LIN {X 0,Y 218.456,Z 624.566,A -85,B 0,C 180,E1 -20246.312,E2 -20246.312} C_VEL
LIN {X 0,Y 218.651,Z 624.551,A -85,B 0,C 180,E1 -20250.001,E2 -20250.001} C_VEL
LIN {X 0,Y 218.485,Z 623.3,A -85,B 0,C 180,E1 -20253.689,E2 -20253.689} C_VEL
LIN {X 0,Y 218.582,Z 620.822,A -85,B 0,C 180,E1 -20257.39,E2 -20257.39} C_VEL
LIN {X 0,Y 219.122,Z 617.082,A -85,B 0,C 180,E1 -20261.096,E2 -20261.096} C_VEL
LIN {X 0,Y 220.229,Z 611.98,A -85,B 0,C 180,E1 -20264.792,E2 -20264.792} C_VEL
LIN {X 0,Y 221.959,Z 605.375,A -85,B 0,C 180,E1 -20268.46,E2 -20268.46} C_VEL
LIN {X 0,Y 224.133,Z 598.233,A -85,B 0,C 180,E1 -20271.619,E2 -20271.619} C_VEL
LIN {X 0,Y 227.018,Z 589.624,A -85,B 0,C 180,E1 -20274.704,E2 -20274.704} C_VEL
LIN {X 0,Y 229.771,Z 580.856,A -85,B 0,C 180,E1 -20277.31,E2 -20277.31} C_VEL
LIN {X 0,Y 233.03,Z 570.467,A -85,B 0,C 180,E1 -20279.843,E2 -20279.843} C_VEL
LIN {X 0,Y 236.861,Z 558.108,A -85,B 0,C 180,E1 -20282.282,E2 -20282.282} C_VEL
LIN {X 0,Y 240.614,Z 544.293,A -85,B 0,C 180,E1 -20284.466,E2 -20284.466} C_VEL
LIN {X 0,Y 243.785,Z 531.6,A -85,B 0,C 180,E1 -20286.06,E2 -20286.06} C_VEL
LIN {X 0,Y 246.726,Z 517.2,A -85,B 0,C 180,E1 -20287.507,E2 -20287.507} C_VEL
LIN {X 0,Y 249.306,Z 502.807,A -85,B 0,C 180,E1 -20288.587,E2 -20288.587} C_VEL
LIN {X 0,Y 251.367,Z 487.341,A -85,B 0,C 180,E1 -20289.434,E2 -20289.434} C_VEL
LIN {X 0,Y 252.647,Z 472.529,A -85,B 0,C 180,E1 -20289.972,E2 -20289.972} C_VEL
LIN {X 0,Y 257.637,Z 382.677,A -85,B 0,C 180,E1 -20292.489,E2 -20292.489} C_VEL
LIN {X 0,Y 249.799,Z 364.197,A -85,B 0,C 180,E1 -20294.587,E2 -20294.587} C_VEL
LIN {X 0,Y 241.793,Z 347.729,A -85,B 0,C 180,E1 -20296.827,E2 -20296.827} C_VEL
LIN {X 0,Y 233.991,Z 333.398,A -85,B 0,C 180,E1 -20299.12,E2 -20299.12} C_VEL
LIN {X 0,Y 227.017,Z 321.467,A -85,B 0,C 180,E1 -20301.335,E2 -20301.335} C_VEL
LIN {X 0,Y 223.588,Z 316.003,A -85,B 0,C 180,E1 -20302.482,E2 -20302.482} C_VEL
LIN {X 0,Y 221.147,Z 311.95,A -85,B 0,C 180,E1 -20303.352,E2 -20303.352} C_VEL
LIN {X 0,Y 220.826,Z 310.593,A -85,B 0,C 180,E1 -20304.067,E2 -20304.067} C_VEL
LIN {X 0,Y 220.813,Z 310.596,A -85,B 0,C 180,E1 -20307.24,E2 -20307.24} C_VEL
LIN {X 0,Y 220.795,Z 310.61,A -85,B 0,C 180,E1 -20311.478,E2 -20311.478} C_VEL
LIN {X 0,Y 220.798,Z 310.607,A -85,B 0,C 180,E1 -20315.554,E2 -20315.554} C_VEL
LIN {X 0,Y 220.849,Z 310.601,A -85,B 0,C 180,E1 -20319.507,E2 -20319.507} C_VEL
LIN {X 0,Y 220.977,Z 310.587,A -85,B 0,C 180,E1 -20323.364,E2 -20323.364} C_VEL
LIN {X 0,Y 221.052,Z 310.539,A -85,B 0,C 180,E1 -20329,E2 -20329} C_VEL
LIN {X 0,Y 221.228,Z 310.552,A -85,B 0,C 180,E1 -20332.697,E2 -20332.697} C_VEL
LIN {X 0,Y 221.432,Z 310.49,A -85,B 0,C 180,E1 -20338.178,E2 -20338.178} C_VEL
LIN {X 0,Y 221.537,Z 310.504,A -85,B 0,C 180,E1 -20339.997,E2 -20339.997} C_VEL
LIN {X 0,Y 221.463,Z 310.523,A -85,B 0,C 180,E1 -20341.816,E2 -20341.816} C_VEL
LIN {X 0,Y 221.209,Z 310.507,A -85,B 0,C 180,E1 -20347.298,E2 -20347.298} C_VEL
LIN {X 0,Y 221.057,Z 310.572,A -85,B 0,C 180,E1 -20350.994,E2 -20350.994} C_VEL
LIN {X 0,Y 220.973,Z 310.534,A -85,B 0,C 180,E1 -20356.63,E2 -20356.63} C_VEL
LIN {X 0,Y 220.862,Z 310.589,A -85,B 0,C 180,E1 -20360.485,E2 -20360.485} C_VEL
LIN {X 0,Y 220.797,Z 310.586,A -85,B 0,C 180,E1 -20364.439,E2 -20364.439} C_VEL
LIN {X 0,Y 220.783,Z 310.569,A -85,B 0,C 180,E1 -20368.517,E2 -20368.517} C_VEL
LIN {X 0,Y 220.802,Z 310.605,A -85,B 0,C 180,E1 -20372.754,E2 -20372.754} C_VEL
LIN {X 0,Y 220.791,Z 310.566,A -85,B 0,C 180,E1 -20377.272,E2 -20377.272} C_VEL
LIN {X 0,Y 220.738,Z 310.614,A -85,B 0,C 180,E1 -20381.955,E2 -20381.955} C_VEL
LIN {X 0,Y 220.751,Z 310.579,A -85,B 0,C 180,E1 -20385.54,E2 -20385.54} C_VEL
LIN {X 0,Y 220.794,Z 310.604,A -85,B 0,C 180,E1 -20390.461,E2 -20390.461} C_VEL
LIN {X 0,Y 220.813,Z 310.578,A -85,B 0,C 180,E1 -20392.791,E2 -20392.791} C_VEL
LIN {X 0,Y 220.802,Z 310.605,A -85,B 0,C 180,E1 -20397.241,E2 -20397.241} C_VEL
LIN {X 0,Y 220.813,Z 310.596,A -85,B 0,C 180,E1 -20401.483,E2 -20401.483} C_VEL
LIN {X 0,Y 220.848,Z 310.585,A -85,B 0,C 180,E1 -20405.563,E2 -20405.563} C_VEL
LIN {X 0,Y 220.859,Z 310.707,A -85,B 0,C 180,E1 -20407.05,E2 -20407.05} C_VEL
LIN {X 0,Y 221.858,Z 313.435,A -85,B 0,C 180,E1 -20407.458,E2 -20407.458} C_VEL
LIN {X 0,Y 224.208,Z 316.191,A -85,B 0,C 180,E1 -20408.217,E2 -20408.217} C_VEL
LIN {X 0,Y 226.521,Z 319.626,A -85,B 0,C 180,E1 -20408.975,E2 -20408.975} C_VEL
LIN {X 0,Y 235.392,Z 332.592,A -85,B 0,C 180,E1 -20411.671,E2 -20411.671} C_VEL
LIN {X 0,Y 247.244,Z 351.934,A -85,B 0,C 180,E1 -20414.953,E2 -20414.953} C_VEL
LIN {X 0,Y 251.217,Z 359.356,A -85,B 0,C 180,E1 -20416,E2 -20416} C_VEL
LIN {X 0,Y 257.92,Z 373.938,A -85,B 0,C 180,E1 -20417.742,E2 -20417.742} C_VEL
LIN {X 0,Y 252.471,Z 467.789,A -85,B 0,C 180,E1 -20420.385,E2 -20420.385} C_VEL
LIN {X 0,Y 250.77,Z 483.73,A -85,B 0,C 180,E1 -20421.133,E2 -20421.133} C_VEL
LIN {X 0,Y 248.657,Z 498.53,A -85,B 0,C 180,E1 -20422.14,E2 -20422.14} C_VEL
LIN {X 0,Y 245.988,Z 512.96,A -85,B 0,C 180,E1 -20423.437,E2 -20423.437} C_VEL
LIN {X 0,Y 243.046,Z 526.643,A -85,B 0,C 180,E1 -20425.023,E2 -20425.023} C_VEL
LIN {X 0,Y 239.557,Z 540.116,A -85,B 0,C 180,E1 -20426.965,E2 -20426.965} C_VEL
LIN {X 0,Y 236.091,Z 552.277,A -85,B 0,C 180,E1 -20429.147,E2 -20429.147} C_VEL
LIN {X 0,Y 232.485,Z 563.947,A -85,B 0,C 180,E1 -20431.732,E2 -20431.732} C_VEL
LIN {X 0,Y 229.373,Z 573.749,A -85,B 0,C 180,E1 -20434.392,E2 -20434.392} C_VEL
LIN {X 0,Y 226.18,Z 583.313,A -85,B 0,C 180,E1 -20437.588,E2 -20437.588} C_VEL
LIN {X 0,Y 223.57,Z 591.227,A -85,B 0,C 180,E1 -20440.871,E2 -20440.871} C_VEL
LIN {X 0,Y 221.829,Z 596.82,A -85,B 0,C 180,E1 -20443.745,E2 -20443.745} C_VEL
LIN {X 0,Y 220.1,Z 602.919,A -85,B 0,C 180,E1 -20447.693,E2 -20447.693} C_VEL
LIN {X 0,Y 219.231,Z 606.386,A -85,B 0,C 180,E1 -20450.647,E2 -20450.647} C_VEL
LIN {X 0,Y 218.41,Z 609.818,A -85,B 0,C 180,E1 -20454.727,E2 -20454.727} C_VEL
LIN {X 0,Y 218.183,Z 610.995,A -85,B 0,C 180,E1 -20456.804,E2 -20456.804} C_VEL
LIN {X 0,Y 218.054,Z 611.981,A -85,B 0,C 180,E1 -20459.523,E2 -20459.523} C_VEL
LIN {X 0,Y 218.223,Z 612.318,A -85,B 0,C 180,E1 -20463.194,E2 -20463.194} C_VEL
LIN {X 0,Y 218.639,Z 611.69,A -85,B 0,C 180,E1 -20466.53,E2 -20466.53} C_VEL
LIN {X 0,Y 219.47,Z 610.095,A -85,B 0,C 180,E1 -20469.823,E2 -20469.823} C_VEL
LIN {X 0,Y 220.653,Z 607.78,A -85,B 0,C 180,E1 -20472.903,E2 -20472.903} C_VEL
LIN {X 0,Y 222.559,Z 603.871,A -85,B 0,C 180,E1 -20476.575,E2 -20476.575} C_VEL
LIN {X 0,Y 224.967,Z 599.012,A -85,B 0,C 180,E1 -20479.938,E2 -20479.938} C_VEL
LIN {X 0,Y 228.653,Z 591.699,A -85,B 0,C 180,E1 -20483.81,E2 -20483.81} C_VEL
LIN {X 0,Y 232.507,Z 583.823,A -85,B 0,C 180,E1 -20487.042,E2 -20487.042} C_VEL
LIN {X 0,Y 237.048,Z 574.291,A -85,B 0,C 180,E1 -20490.132,E2 -20490.132} C_VEL
LIN {X 0,Y 241.578,Z 564.062,A -85,B 0,C 180,E1 -20492.789,E2 -20492.789} C_VEL
LIN {X 0,Y 246.371,Z 552.376,A -85,B 0,C 180,E1 -20495.215,E2 -20495.215} C_VEL
LIN {X 0,Y 251.205,Z 539.173,A -85,B 0,C 180,E1 -20497.4,E2 -20497.4} C_VEL
LIN {X 0,Y 255.148,Z 527.022,A -85,B 0,C 180,E1 -20499.021,E2 -20499.021} C_VEL
LIN {X 0,Y 259.043,Z 512.878,A -85,B 0,C 180,E1 -20500.52,E2 -20500.52} C_VEL
LIN {X 0,Y 262.341,Z 498.015,A -85,B 0,C 180,E1 -20501.742,E2 -20501.742} C_VEL
LIN {X 0,Y 265.039,Z 482.598,A -85,B 0,C 180,E1 -20502.664,E2 -20502.664} C_VEL
LIN {X 0,Y 266.874,Z 468.107,A -85,B 0,C 180,E1 -20503.265,E2 -20503.265} C_VEL
LIN {X 0,Y 273.007,Z 383.244,A -85,B 0,C 180,E1 -20505.604,E2 -20505.604} C_VEL
LIN {X 0,Y 267.895,Z 372.276,A -85,B 0,C 180,E1 -20507.64,E2 -20507.64} C_VEL
LIN {X 0,Y 263.593,Z 364.08,A -85,B 0,C 180,E1 -20509.487,E2 -20509.487} C_VEL
LIN {X 0,Y 258.502,Z 356.176,A -85,B 0,C 180,E1 -20511.83,E2 -20511.83} C_VEL
LIN {X 0,Y 254.898,Z 351,A -85,B 0,C 180,E1 -20513.671,E2 -20513.671} C_VEL
LIN {X 0,Y 252.726,Z 347.79,A -85,B 0,C 180,E1 -20514.896,E2 -20514.896} C_VEL
LIN {X 0,Y 250.186,Z 344.212,A -85,B 0,C 180,E1 -20516.453,E2 -20516.453} C_VEL
LIN {X 0,Y 247.433,Z 340.87,A -85,B 0,C 180,E1 -20518.278,E2 -20518.278} C_VEL
LIN {X 0,Y 246.259,Z 338.983,A -85,B 0,C 180,E1 -20519.185,E2 -20519.185} C_VEL
LIN {X 0,Y 243.713,Z 335.653,A -85,B 0,C 180,E1 -20521.321,E2 -20521.321} C_VEL
LIN {X 0,Y 242.954,Z 334.278,A -85,B 0,C 180,E1 -20522.075,E2 -20522.075} C_VEL
LIN {X 0,Y 240.47,Z 332.623,A -85,B 0,C 180,E1 -20524.515,E2 -20524.515} C_VEL
LIN {X 0,Y 239.323,Z 332.075,A -85,B 0,C 180,E1 -20525.898,E2 -20525.898} C_VEL
LIN {X 0,Y 237.497,Z 333.141,A -85,B 0,C 180,E1 -20528.234,E2 -20528.234} C_VEL
LIN {X 0,Y 235.878,Z 334.987,A -85,B 0,C 180,E1 -20531.099,E2 -20531.099} C_VEL
LIN {X 0,Y 235.577,Z 335.118,A -85,B 0,C 180,E1 -20532.072,E2 -20532.072} C_VEL
LIN {X 0,Y 235.39,Z 335.075,A -85,B 0,C 180,E1 -20536.649,E2 -20536.649} C_VEL
LIN {X 0,Y 237.107,Z 336.043,A -85,B 0,C 180,E1 -20541.447,E2 -20541.447} C_VEL
LIN {X 0,Y 238.494,Z 338.96,A -85,B 0,C 180,E1 -20543.906,E2 -20543.906} C_VEL
LIN {X 0,Y 240.684,Z 341.484,A -85,B 0,C 180,E1 -20546.504,E2 -20546.504} C_VEL
LIN {X 0,Y 242.423,Z 343.819,A -85,B 0,C 180,E1 -20548.221,E2 -20548.221} C_VEL
LIN {X 0,Y 246.306,Z 349.812,A -85,B 0,C 180,E1 -20551.463,E2 -20551.463} C_VEL
LIN {X 0,Y 249.599,Z 355.143,A -85,B 0,C 180,E1 -20553.723,E2 -20553.723} C_VEL
LIN {X 0,Y 253.215,Z 361.416,A -85,B 0,C 180,E1 -20555.918,E2 -20555.918} C_VEL
LIN {X 0,Y 257.045,Z 368.192,A -85,B 0,C 180,E1 -20557.967,E2 -20557.967} C_VEL
LIN {X 0,Y 261.448,Z 377.097,A -85,B 0,C 180,E1 -20560.122,E2 -20560.122} C_VEL
LIN {X 0,Y 265.545,Z 386.333,A -85,B 0,C 180,E1 -20561.978,E2 -20561.978} C_VEL
LIN {X 0,Y 268.211,Z 392.988,A -85,B 0,C 180,E1 -20563.118,E2 -20563.118} C_VEL
LIN {X 0,Y 262.753,Z 466.073,A -85,B 0,C 180,E1 -20565.118,E2 -20565.118} C_VEL
LIN {X 0,Y 261.154,Z 482.947,A -85,B 0,C 180,E1 -20565.667,E2 -20565.667} C_VEL
LIN {X 0,Y 258.786,Z 498.008,A -85,B 0,C 180,E1 -20566.374,E2 -20566.374} C_VEL
LIN {X 0,Y 255.719,Z 512.24,A -85,B 0,C 180,E1 -20567.276,E2 -20567.276} C_VEL
LIN {X 0,Y 252.391,Z 524.954,A -85,B 0,C 180,E1 -20568.334,E2 -20568.334} C_VEL
LIN {X 0,Y 248.42,Z 538.188,A -85,B 0,C 180,E1 -20569.761,E2 -20569.761} C_VEL
LIN {X 0,Y 243.97,Z 550.9,A -85,B 0,C 180,E1 -20571.47,E2 -20571.47} C_VEL
LIN {X 0,Y 239.283,Z 562.966,A -85,B 0,C 180,E1 -20573.506,E2 -20573.506} C_VEL
LIN {X 0,Y 234.433,Z 574.046,A -85,B 0,C 180,E1 -20575.801,E2 -20575.801} C_VEL
LIN {X 0,Y 229.392,Z 584.891,A -85,B 0,C 180,E1 -20578.613,E2 -20578.613} C_VEL
LIN {X 0,Y 225.022,Z 594.02,A -85,B 0,C 180,E1 -20581.588,E2 -20581.588} C_VEL
LIN {X 0,Y 221.182,Z 601.509,A -85,B 0,C 180,E1 -20584.6,E2 -20584.6} C_VEL
LIN {X 0,Y 217.655,Z 608.62,A -85,B 0,C 180,E1 -20588.204,E2 -20588.204} C_VEL
LIN {X 0,Y 214.881,Z 614.415,A -85,B 0,C 180,E1 -20592.007,E2 -20592.007} C_VEL
LIN {X 0,Y 213.495,Z 617.698,A -85,B 0,C 180,E1 -20594.732,E2 -20594.732} C_VEL
LIN {X 0,Y 212.119,Z 621.093,A -85,B 0,C 180,E1 -20598.535,E2 -20598.535} C_VEL
LIN {X 0,Y 211.489,Z 623.304,A -85,B 0,C 180,E1 -20602.362,E2 -20602.362} C_VEL
LIN {X 0,Y 211.355,Z 624.375,A -85,B 0,C 180,E1 -20606.188,E2 -20606.188} C_VEL
LIN {X 0,Y 211.567,Z 624.306,A -85,B 0,C 180,E1 -20610.001,E2 -20610.001} C_VEL
LIN {X 0,Y 211.404,Z 623.029,A -85,B 0,C 180,E1 -20613.813,E2 -20613.813} C_VEL
LIN {X 0,Y 211.51,Z 620.495,A -85,B 0,C 180,E1 -20617.638,E2 -20617.638} C_VEL
LIN {X 0,Y 212.096,Z 616.695,A -85,B 0,C 180,E1 -20621.468,E2 -20621.468} C_VEL
LIN {X 0,Y 213.277,Z 611.528,A -85,B 0,C 180,E1 -20625.285,E2 -20625.285} C_VEL
LIN {X 0,Y 215.164,Z 604.857,A -85,B 0,C 180,E1 -20629.065,E2 -20629.065} C_VEL
LIN {X 0,Y 217.447,Z 597.637,A -85,B 0,C 180,E1 -20632.32,E2 -20632.32} C_VEL
LIN {X 0,Y 220.52,Z 588.944,A -85,B 0,C 180,E1 -20635.483,E2 -20635.483} C_VEL
LIN {X 0,Y 223.868,Z 578.579,A -85,B 0,C 180,E1 -20638.552,E2 -20638.552} C_VEL
LIN {X 0,Y 227.437,Z 567.62,A -85,B 0,C 180,E1 -20641.171,E2 -20641.171} C_VEL
LIN {X 0,Y 231.11,Z 555.864,A -85,B 0,C 180,E1 -20643.448,E2 -20643.448} C_VEL
LIN {X 0,Y 234.703,Z 543.03,A -85,B 0,C 180,E1 -20645.462,E2 -20645.462} C_VEL
LIN {X 0,Y 238.13,Z 529.368,A -85,B 0,C 180,E1 -20647.166,E2 -20647.166} C_VEL
LIN {X 0,Y 241.119,Z 515.359,A -85,B 0,C 180,E1 -20648.537,E2 -20648.537} C_VEL
LIN {X 0,Y 243.645,Z 501.196,A -85,B 0,C 180,E1 -20649.59,E2 -20649.59} C_VEL
LIN {X 0,Y 245.656,Z 486.133,A -85,B 0,C 180,E1 -20650.404,E2 -20650.404} C_VEL
LIN {X 0,Y 246.926,Z 470.859,A -85,B 0,C 180,E1 -20650.956,E2 -20650.956} C_VEL
LIN {X 0,Y 251.89,Z 384.671,A -85,B 0,C 180,E1 -20653.408,E2 -20653.408} C_VEL
LIN {X 0,Y 243.631,Z 365.283,A -85,B 0,C 180,E1 -20655.723,E2 -20655.723} C_VEL
LIN {X 0,Y 234.754,Z 347.393,A -85,B 0,C 180,E1 -20658.328,E2 -20658.328} C_VEL
LIN {X 0,Y 226.161,Z 331.72,A -85,B 0,C 180,E1 -20661.059,E2 -20661.059} C_VEL
LIN {X 0,Y 219.322,Z 320.59,A -85,B 0,C 180,E1 -20663.381,E2 -20663.381} C_VEL
LIN {X 0,Y 216.365,Z 316.114,A -85,B 0,C 180,E1 -20664.432,E2 -20664.432} C_VEL
LIN {X 0,Y 214.484,Z 313.799,A -85,B 0,C 180,E1 -20665.098,E2 -20665.098} C_VEL
LIN {X 0,Y 213.759,Z 311.528,A -85,B 0,C 180,E1 -20665.518,E2 -20665.518} C_VEL
LIN {X 0,Y 213.772,Z 311.48,A -85,B 0,C 180,E1 -20668.735,E2 -20668.735} C_VEL
LIN {X 0,Y 213.769,Z 311.477,A -85,B 0,C 180,E1 -20672.592,E2 -20672.592} C_VEL
LIN {X 0,Y 213.782,Z 311.479,A -85,B 0,C 180,E1 -20676.997,E2 -20676.997} C_VEL
LIN {X 0,Y 213.885,Z 311.473,A -85,B 0,C 180,E1 -20682.796,E2 -20682.796} C_VEL
LIN {X 0,Y 213.922,Z 311.416,A -85,B 0,C 180,E1 -20686.702,E2 -20686.702} C_VEL
LIN {X 0,Y 214.123,Z 311.426,A -85,B 0,C 180,E1 -20690.551,E2 -20690.551} C_VEL
LIN {X 0,Y 214.061,Z 311.423,A -85,B 0,C 180,E1 -20694.344,E2 -20694.344} C_VEL
LIN {X 0,Y 214.372,Z 311.367,A -85,B 0,C 180,E1 -20698.118,E2 -20698.118} C_VEL
LIN {X 0,Y 214.505,Z 311.379,A -85,B 0,C 180,E1 -20699.997,E2 -20699.997} C_VEL
LIN {X 0,Y 214.4,Z 311.403,A -85,B 0,C 180,E1 -20701.875,E2 -20701.875} C_VEL
LIN {X 0,Y 214.153,Z 311.386,A -85,B 0,C 180,E1 -20707.54,E2 -20707.54} C_VEL
LIN {X 0,Y 213.988,Z 311.455,A -85,B 0,C 180,E1 -20711.362,E2 -20711.362} C_VEL
LIN {X 0,Y 213.895,Z 311.426,A -85,B 0,C 180,E1 -20715.236,E2 -20715.236} C_VEL
LIN {X 0,Y 213.799,Z 311.447,A -85,B 0,C 180,E1 -20719.187,E2 -20719.187} C_VEL
LIN {X 0,Y 213.779,Z 311.475,A -85,B 0,C 180,E1 -20723.231,E2 -20723.231} C_VEL
LIN {X 0,Y 213.759,Z 311.435,A -85,B 0,C 180,E1 -20727.414,E2 -20727.414} C_VEL
LIN {X 0,Y 213.75,Z 311.485,A -85,B 0,C 180,E1 -20731.736,E2 -20731.736} C_VEL
LIN {X 0,Y 213.732,Z 311.444,A -85,B 0,C 180,E1 -20736.286,E2 -20736.286} C_VEL
LIN {X 0,Y 213.688,Z 311.495,A -85,B 0,C 180,E1 -20741.126,E2 -20741.126} C_VEL
LIN {X 0,Y 213.691,Z 311.469,A -85,B 0,C 180,E1 -20743.677,E2 -20743.677} C_VEL
LIN {X 0,Y 213.692,Z 311.461,A -85,B 0,C 180,E1 -20746.342,E2 -20746.342} C_VEL
LIN {X 0,Y 213.705,Z 311.495,A -85,B 0,C 180,E1 -20749.141,E2 -20749.141} C_VEL
LIN {X 0,Y 213.729,Z 311.462,A -85,B 0,C 180,E1 -20753.709,E2 -20753.709} C_VEL
LIN {X 0,Y 213.755,Z 311.467,A -85,B 0,C 180,E1 -20758.26,E2 -20758.26} C_VEL
LIN {X 0,Y 213.814,Z 311.478,A -85,B 0,C 180,E1 -20762.601,E2 -20762.601} C_VEL
LIN {X 0,Y 213.811,Z 311.46,A -85,B 0,C 180,E1 -20765.089,E2 -20765.089} C_VEL
LIN {X 0,Y 214.689,Z 314.123,A -85,B 0,C 180,E1 -20765.497,E2 -20765.497} C_VEL
LIN {X 0,Y 217.186,Z 317.07,A -85,B 0,C 180,E1 -20766.364,E2 -20766.364} C_VEL
LIN {X 0,Y 219.257,Z 320.248,A -85,B 0,C 180,E1 -20767.1,E2 -20767.1} C_VEL
LIN {X 0,Y 220.544,Z 321.783,A -85,B 0,C 180,E1 -20767.527,E2 -20767.527} C_VEL
LIN {X 0,Y 231.141,Z 337.351,A -85,B 0,C 180,E1 -20770.915,E2 -20770.915} C_VEL
LIN {X 0,Y 242.343,Z 355.847,A -85,B 0,C 180,E1 -20774.144,E2 -20774.144} C_VEL
LIN {X 0,Y 246.211,Z 363.031,A -85,B 0,C 180,E1 -20775.203,E2 -20775.203} C_VEL
LIN {X 0,Y 252.216,Z 376.176,A -85,B 0,C 180,E1 -20776.837,E2 -20776.837} C_VEL
LIN {X 0,Y 246.709,Z 467.338,A -85,B 0,C 180,E1 -20779.433,E2 -20779.433} C_VEL
LIN {X 0,Y 244.943,Z 483.516,A -85,B 0,C 180,E1 -20780.191,E2 -20780.191} C_VEL
LIN {X 0,Y 242.68,Z 498.892,A -85,B 0,C 180,E1 -20781.254,E2 -20781.254} C_VEL
LIN {X 0,Y 240.197,Z 512.019,A -85,B 0,C 180,E1 -20782.44,E2 -20782.44} C_VEL
LIN {X 0,Y 237.142,Z 525.879,A -85,B 0,C 180,E1 -20784.046,E2 -20784.046} C_VEL
LIN {X 0,Y 233.733,Z 538.791,A -85,B 0,C 180,E1 -20785.904,E2 -20785.904} C_VEL
LIN {X 0,Y 229.938,Z 551.825,A -85,B 0,C 180,E1 -20788.248,E2 -20788.248} C_VEL
LIN {X 0,Y 226.173,Z 563.617,A -85,B 0,C 180,E1 -20790.889,E2 -20790.889} C_VEL
LIN {X 0,Y 222.901,Z 573.498,A -85,B 0,C 180,E1 -20793.615,E2 -20793.615} C_VEL
LIN {X 0,Y 219.473,Z 583.348,A -85,B 0,C 180,E1 -20796.967,E2 -20796.967} C_VEL
LIN {X 0,Y 216.797,Z 591.135,A -85,B 0,C 180,E1 -20800.27,E2 -20800.27} C_VEL
LIN {X 0,Y 214.972,Z 596.767,A -85,B 0,C 180,E1 -20803.228,E2 -20803.228} C_VEL
LIN {X 0,Y 213.136,Z 602.878,A -85,B 0,C 180,E1 -20807.262,E2 -20807.262} C_VEL
LIN {X 0,Y 212.222,Z 606.445,A -85,B 0,C 180,E1 -20810.347,E2 -20810.347} C_VEL
LIN {X 0,Y 211.471,Z 609.197,A -85,B 0,C 180,E1 -20813.502,E2 -20813.502} C_VEL
LIN {X 0,Y 211.145,Z 610.816,A -85,B 0,C 180,E1 -20816.022,E2 -20816.022} C_VEL
LIN {X 0,Y 210.961,Z 612.273,A -85,B 0,C 180,E1 -20819.992,E2 -20819.992} C_VEL
LIN {X 0,Y 211.162,Z 612.512,A -85,B 0,C 180,E1 -20823.696,E2 -20823.696} C_VEL
LIN {X 0,Y 211.652,Z 611.805,A -85,B 0,C 180,E1 -20827.169,E2 -20827.169} C_VEL
LIN {X 0,Y 212.881,Z 609.688,A -85,B 0,C 180,E1 -20831.319,E2 -20831.319} C_VEL
LIN {X 0,Y 214.443,Z 606.8,A -85,B 0,C 180,E1 -20834.796,E2 -20834.796} C_VEL
LIN {X 0,Y 217.054,Z 601.8,A -85,B 0,C 180,E1 -20839.039,E2 -20839.039} C_VEL
LIN {X 0,Y 220.376,Z 595.616,A -85,B 0,C 180,E1 -20842.868,E2 -20842.868} C_VEL
LIN {X 0,Y 224.225,Z 588.37,A -85,B 0,C 180,E1 -20846.312,E2 -20846.312} C_VEL
LIN {X 0,Y 228.488,Z 580.005,A -85,B 0,C 180,E1 -20849.453,E2 -20849.453} C_VEL
LIN {X 0,Y 232.711,Z 571.395,A -85,B 0,C 180,E1 -20852.047,E2 -20852.047} C_VEL
LIN {X 0,Y 237.359,Z 561.234,A -85,B 0,C 180,E1 -20854.562,E2 -20854.562} C_VEL
LIN {X 0,Y 241.956,Z 550.246,A -85,B 0,C 180,E1 -20856.768,E2 -20856.768} C_VEL
LIN {X 0,Y 246.645,Z 537.72,A -85,B 0,C 180,E1 -20858.798,E2 -20858.798} C_VEL
LIN {X 0,Y 251.213,Z 523.82,A -85,B 0,C 180,E1 -20860.573,E2 -20860.573} C_VEL
LIN {X 0,Y 254.929,Z 510.143,A -85,B 0,C 180,E1 -20861.96,E2 -20861.96} C_VEL
LIN {X 0,Y 258.058,Z 496.201,A -85,B 0,C 180,E1 -20863.051,E2 -20863.051} C_VEL
LIN {X 0,Y 260.673,Z 481.287,A -85,B 0,C 180,E1 -20863.92,E2 -20863.92} C_VEL
LIN {X 0,Y 262.54,Z 466.44,A -85,B 0,C 180,E1 -20864.506,E2 -20864.506} C_VEL
LIN {X 0,Y 268.549,Z 386.105,A -85,B 0,C 180,E1 -20866.747,E2 -20866.747} C_VEL
LIN {X 0,Y 264.25,Z 376.744,A -85,B 0,C 180,E1 -20868.571,E2 -20868.571} C_VEL
LIN {X 0,Y 260.856,Z 370.046,A -85,B 0,C 180,E1 -20870.111,E2 -20870.111} C_VEL
LIN {X 0,Y 255.935,Z 362.078,A -85,B 0,C 180,E1 -20872.499,E2 -20872.499} C_VEL
LIN {X 0,Y 250.767,Z 354.287,A -85,B 0,C 180,E1 -20875.376,E2 -20875.376} C_VEL
LIN {X 0,Y 248.058,Z 350.485,A -85,B 0,C 180,E1 -20877.098,E2 -20877.098} C_VEL
LIN {X 0,Y 245.244,Z 346.709,A -85,B 0,C 180,E1 -20879.112,E2 -20879.112} C_VEL
LIN {X 0,Y 244.278,Z 345.307,A -85,B 0,C 180,E1 -20879.881,E2 -20879.881} C_VEL
LIN {X 0,Y 241.865,Z 341.734,A -85,B 0,C 180,E1 -20882.084,E2 -20882.084} C_VEL
LIN {X 0,Y 241.22,Z 340.961,A -85,B 0,C 180,E1 -20882.716,E2 -20882.716} C_VEL
LIN {X 0,Y 238.566,Z 338.718,A -85,B 0,C 180,E1 -20885.673,E2 -20885.673} C_VEL
LIN {X 0,Y 237.351,Z 335.924,A -85,B 0,C 180,E1 -20887.82,E2 -20887.82} C_VEL
LIN {X 0,Y 235.577,Z 335.118,A -85,B 0,C 180,E1 -20892.072,E2 -20892.072} C_VEL
LIN {X 0,Y 235.237,Z 335.683,A -85,B 0,C 180,E1 -20893.5,E2 -20893.5} C_VEL
LIN {X 0,Y 234.791,Z 338.536,A -85,B 0,C 180,E1 -20895.813,E2 -20895.813} C_VEL
LIN {X 0,Y 234.767,Z 341.115,A -85,B 0,C 180,E1 -20897.659,E2 -20897.659} C_VEL
LIN {X 0,Y 235.025,Z 342.388,A -85,B 0,C 180,E1 -20899.077,E2 -20899.077} C_VEL
LIN {X 0,Y 235.194,Z 342.576,A -85,B 0,C 180,E1 -20899.556,E2 -20899.556} C_VEL
LIN {X 0,Y 235.948,Z 343.065,A -85,B 0,C 180,E1 -20901.175,E2 -20901.175} C_VEL
LIN {X 0,Y 237.766,Z 346.541,A -85,B 0,C 180,E1 -20904.305,E2 -20904.305} C_VEL
LIN {X 0,Y 239.31,Z 348.277,A -85,B 0,C 180,E1 -20906.139,E2 -20906.139} C_VEL
LIN {X 0,Y 240.834,Z 350.436,A -85,B 0,C 180,E1 -20907.721,E2 -20907.721} C_VEL
LIN {X 0,Y 244.554,Z 356.398,A -85,B 0,C 180,E1 -20910.977,E2 -20910.977} C_VEL
LIN {X 0,Y 247.446,Z 361.331,A -85,B 0,C 180,E1 -20913.081,E2 -20913.081} C_VEL
LIN {X 0,Y 251.269,Z 368.202,A -85,B 0,C 180,E1 -20915.514,E2 -20915.514} C_VEL
LIN {X 0,Y 254.91,Z 375.131,A -85,B 0,C 180,E1 -20917.543,E2 -20917.543} C_VEL
LIN {X 0,Y 258.707,Z 383.185,A -85,B 0,C 180,E1 -20919.496,E2 -20919.496} C_VEL
LIN {X 0,Y 262.482,Z 392.088,A -85,B 0,C 180,E1 -20921.299,E2 -20921.299} C_VEL
LIN {X 0,Y 263.915,Z 395.738,A -85,B 0,C 180,E1 -20921.956,E2 -20921.956} C_VEL
LIN {X 0,Y 257.431,Z 477.529,A -85,B 0,C 180,E1 -20924.225,E2 -20924.225} C_VEL
LIN {X 0,Y 255.144,Z 493.475,A -85,B 0,C 180,E1 -20924.895,E2 -20924.895} C_VEL
LIN {X 0,Y 251.968,Z 508.72,A -85,B 0,C 180,E1 -20925.791,E2 -20925.791} C_VEL
LIN {X 0,Y 248.249,Z 522.941,A -85,B 0,C 180,E1 -20926.925,E2 -20926.925} C_VEL
LIN {X 0,Y 243.735,Z 537.416,A -85,B 0,C 180,E1 -20928.458,E2 -20928.458} C_VEL
LIN {X 0,Y 238.943,Z 550.581,A -85,B 0,C 180,E1 -20930.23,E2 -20930.23} C_VEL
LIN {X 0,Y 234.492,Z 561.635,A -85,B 0,C 180,E1 -20932.093,E2 -20932.093} C_VEL
LIN {X 0,Y 229.429,Z 572.873,A -85,B 0,C 180,E1 -20934.409,E2 -20934.409} C_VEL
LIN {X 0,Y 224.773,Z 582.39,A -85,B 0,C 180,E1 -20936.828,E2 -20936.828} C_VEL
LIN {X 0,Y 220.052,Z 591.625,A -85,B 0,C 180,E1 -20939.729,E2 -20939.729} C_VEL
LIN {X 0,Y 215.901,Z 599.683,A -85,B 0,C 180,E1 -20942.89,E2 -20942.89} C_VEL
LIN {X 0,Y 211.879,Z 607.115,A -85,B 0,C 180,E1 -20946.546,E2 -20946.546} C_VEL
LIN {X 0,Y 208.728,Z 613.057,A -85,B 0,C 180,E1 -20950.325,E2 -20950.325} C_VEL
LIN {X 0,Y 206.601,Z 617.671,A -85,B 0,C 180,E1 -20954.21,E2 -20954.21} C_VEL
LIN {X 0,Y 205.118,Z 621.02,A -85,B 0,C 180,E1 -20958.138,E2 -20958.138} C_VEL
LIN {X 0,Y 204.422,Z 623.172,A -85,B 0,C 180,E1 -20962.097,E2 -20962.097} C_VEL
LIN {X 0,Y 204.267,Z 624.199,A -85,B 0,C 180,E1 -20966.206,E2 -20966.206} C_VEL
LIN {X 0,Y 204.483,Z 624.056,A -85,B 0,C 180,E1 -20970.001,E2 -20970.001} C_VEL
LIN {X 0,Y 204.329,Z 622.68,A -85,B 0,C 180,E1 -20974.045,E2 -20974.045} C_VEL
LIN {X 0,Y 204.44,Z 620.155,A -85,B 0,C 180,E1 -20977.904,E2 -20977.904} C_VEL
LIN {X 0,Y 205.064,Z 616.288,A -85,B 0,C 180,E1 -20981.867,E2 -20981.867} C_VEL
LIN {X 0,Y 206.345,Z 611.05,A -85,B 0,C 180,E1 -20985.812,E2 -20985.812} C_VEL
LIN {X 0,Y 208.384,Z 604.301,A -85,B 0,C 180,E1 -20989.711,E2 -20989.711} C_VEL
LIN {X 0,Y 210.795,Z 596.992,A -85,B 0,C 180,E1 -20993.064,E2 -20993.064} C_VEL
LIN {X 0,Y 214.054,Z 588.204,A -85,B 0,C 180,E1 -20996.311,E2 -20996.311} C_VEL
LIN {X 0,Y 217.645,Z 577.562,A -85,B 0,C 180,E1 -20999.501,E2 -20999.501} C_VEL
LIN {X 0,Y 221.3,Z 566.637,A -85,B 0,C 180,E1 -21002.137,E2 -21002.137} C_VEL
LIN {X 0,Y 225.145,Z 554.725,A -85,B 0,C 180,E1 -21004.456,E2 -21004.456} C_VEL
LIN {X 0,Y 228.857,Z 541.684,A -85,B 0,C 180,E1 -21006.512,E2 -21006.512} C_VEL
LIN {X 0,Y 232.332,Z 528.152,A -85,B 0,C 180,E1 -21008.196,E2 -21008.196} C_VEL
LIN {X 0,Y 235.555,Z 513.382,A -85,B 0,C 180,E1 -21009.624,E2 -21009.624} C_VEL
LIN {X 0,Y 238.189,Z 498.634,A -85,B 0,C 180,E1 -21010.685,E2 -21010.685} C_VEL
LIN {X 0,Y 240.121,Z 483.561,A -85,B 0,C 180,E1 -21011.468,E2 -21011.468} C_VEL
LIN {X 0,Y 241.559,Z 464.185,A -85,B 0,C 180,E1 -21012.12,E2 -21012.12} C_VEL
LIN {X 0,Y 246.164,Z 386.755,A -85,B 0,C 180,E1 -21014.363,E2 -21014.363} C_VEL
LIN {X 0,Y 238.799,Z 369.227,A -85,B 0,C 180,E1 -21016.53,E2 -21016.53} C_VEL
LIN {X 0,Y 229.874,Z 351.032,A -85,B 0,C 180,E1 -21019.263,E2 -21019.263} C_VEL
LIN {X 0,Y 221.88,Z 336.336,A -85,B 0,C 180,E1 -21021.917,E2 -21021.917} C_VEL
LIN {X 0,Y 215.068,Z 325.068,A -85,B 0,C 180,E1 -21024.33,E2 -21024.33} C_VEL
LIN {X 0,Y 212.842,Z 321.745,A -85,B 0,C 180,E1 -21025.155,E2 -21025.155} C_VEL
LIN {X 0,Y 210.577,Z 318.68,A -85,B 0,C 180,E1 -21026.008,E2 -21026.008} C_VEL
LIN {X 0,Y 209.71,Z 317.316,A -85,B 0,C 180,E1 -21026.354,E2 -21026.354} C_VEL
LIN {X 0,Y 207.648,Z 315.113,A -85,B 0,C 180,E1 -21027.137,E2 -21027.137} C_VEL
LIN {X 0,Y 206.762,Z 312.798,A -85,B 0,C 180,E1 -21027.558,E2 -21027.558} C_VEL
LIN {X 0,Y 206.689,Z 312.36,A -85,B 0,C 180,E1 -21027.684,E2 -21027.684} C_VEL
LIN {X 0,Y 206.699,Z 312.36,A -85,B 0,C 180,E1 -21032.132,E2 -21032.132} C_VEL
LIN {X 0,Y 206.712,Z 312.358,A -85,B 0,C 180,E1 -21036.63,E2 -21036.63} C_VEL
LIN {X 0,Y 206.805,Z 312.355,A -85,B 0,C 180,E1 -21042.187,E2 -21042.187} C_VEL
LIN {X 0,Y 206.863,Z 312.298,A -85,B 0,C 180,E1 -21046.239,E2 -21046.239} C_VEL
LIN {X 0,Y 207.072,Z 312.299,A -85,B 0,C 180,E1 -21050.227,E2 -21050.227} C_VEL
LIN {X 0,Y 207.026,Z 312.302,A -85,B 0,C 180,E1 -21054.152,E2 -21054.152} C_VEL
LIN {X 0,Y 207.314,Z 312.245,A -85,B 0,C 180,E1 -21058.054,E2 -21058.054} C_VEL
LIN {X 0,Y 207.473,Z 312.255,A -85,B 0,C 180,E1 -21059.997,E2 -21059.997} C_VEL
LIN {X 0,Y 207.339,Z 312.282,A -85,B 0,C 180,E1 -21061.939,E2 -21061.939} C_VEL
LIN {X 0,Y 207.101,Z 312.266,A -85,B 0,C 180,E1 -21067.798,E2 -21067.798} C_VEL
LIN {X 0,Y 206.911,Z 312.337,A -85,B 0,C 180,E1 -21071.756,E2 -21071.756} C_VEL
LIN {X 0,Y 206.822,Z 312.3,A -85,B 0,C 180,E1 -21075.771,E2 -21075.771} C_VEL
LIN {X 0,Y 206.719,Z 312.34,A -85,B 0,C 180,E1 -21079.872,E2 -21079.872} C_VEL
LIN {X 0,Y 206.692,Z 312.347,A -85,B 0,C 180,E1 -21084.077,E2 -21084.077} C_VEL
LIN {X 0,Y 206.67,Z 312.323,A -85,B 0,C 180,E1 -21088.426,E2 -21088.426} C_VEL
LIN {X 0,Y 206.685,Z 312.361,A -85,B 0,C 180,E1 -21092.956,E2 -21092.956} C_VEL
LIN {X 0,Y 206.691,Z 312.327,A -85,B 0,C 180,E1 -21095.308,E2 -21095.308} C_VEL
LIN {X 0,Y 206.637,Z 312.368,A -85,B 0,C 180,E1 -21100.252,E2 -21100.252} C_VEL
LIN {X 0,Y 206.619,Z 312.341,A -85,B 0,C 180,E1 -21104.414,E2 -21104.414} C_VEL
LIN {X 0,Y 206.629,Z 312.37,A -85,B 0,C 180,E1 -21108.435,E2 -21108.435} C_VEL
LIN {X 0,Y 206.661,Z 312.342,A -85,B 0,C 180,E1 -21112.256,E2 -21112.256} C_VEL
LIN {X 0,Y 206.685,Z 312.364,A -85,B 0,C 180,E1 -21117.04,E2 -21117.04} C_VEL
LIN {X 0,Y 206.752,Z 312.356,A -85,B 0,C 180,E1 -21122.096,E2 -21122.096} C_VEL
LIN {X 0,Y 206.789,Z 312.495,A -85,B 0,C 180,E1 -21122.962,E2 -21122.962} C_VEL
LIN {X 0,Y 207.614,Z 314.959,A -85,B 0,C 180,E1 -21123.373,E2 -21123.373} C_VEL
LIN {X 0,Y 209.533,Z 317.168,A -85,B 0,C 180,E1 -21124.107,E2 -21124.107} C_VEL
LIN {X 0,Y 210.291,Z 318.034,A -85,B 0,C 180,E1 -21124.392,E2 -21124.392} C_VEL
LIN {X 0,Y 212.49,Z 321.34,A -85,B 0,C 180,E1 -21125.239,E2 -21125.239} C_VEL
LIN {X 0,Y 213.851,Z 323.196,A -85,B 0,C 180,E1 -21125.738,E2 -21125.738} C_VEL
LIN {X 0,Y 217.333,Z 328.028,A -85,B 0,C 180,E1 -21126.971,E2 -21126.971} C_VEL
LIN {X 0,Y 225.406,Z 339.932,A -85,B 0,C 180,E1 -21129.669,E2 -21129.669} C_VEL
LIN {X 0,Y 234.865,Z 355.293,A -85,B 0,C 180,E1 -21132.561,E2 -21132.561} C_VEL
LIN {X 0,Y 241.359,Z 366.943,A -85,B 0,C 180,E1 -21134.407,E2 -21134.407} C_VEL
LIN {X 0,Y 246.513,Z 378.667,A -85,B 0,C 180,E1 -21135.892,E2 -21135.892} C_VEL
LIN {X 0,Y 240.908,Z 467.99,A -85,B 0,C 180,E1 -21138.483,E2 -21138.483} C_VEL
LIN {X 0,Y 239.091,Z 483.988,A -85,B 0,C 180,E1 -21139.253,E2 -21139.253} C_VEL
LIN {X 0,Y 236.865,Z 498.707,A -85,B 0,C 180,E1 -21140.284,E2 -21140.284} C_VEL
LIN {X 0,Y 234.104,Z 512.804,A -85,B 0,C 180,E1 -21141.584,E2 -21141.584} C_VEL
LIN {X 0,Y 230.92,Z 526.616,A -85,B 0,C 180,E1 -21143.227,E2 -21143.227} C_VEL
LIN {X 0,Y 227.424,Z 539.436,A -85,B 0,C 180,E1 -21145.124,E2 -21145.124} C_VEL
LIN {X 0,Y 223.482,Z 552.386,A -85,B 0,C 180,E1 -21147.521,E2 -21147.521} C_VEL
LIN {X 0,Y 219.91,Z 563.223,A -85,B 0,C 180,E1 -21149.999,E2 -21149.999} C_VEL
LIN {X 0,Y 216.464,Z 573.186,A -85,B 0,C 180,E1 -21152.791,E2 -21152.791} C_VEL
LIN {X 0,Y 213.409,Z 581.63,A -85,B 0,C 180,E1 -21155.669,E2 -21155.669} C_VEL
LIN {X 0,Y 210.414,Z 589.908,A -85,B 0,C 180,E1 -21159.128,E2 -21159.128} C_VEL
LIN {X 0,Y 208.039,Z 596.907,A -85,B 0,C 180,E1 -21162.807,E2 -21162.807} C_VEL
LIN {X 0,Y 206.589,Z 601.502,A -85,B 0,C 180,E1 -21165.791,E2 -21165.791} C_VEL
LIN {X 0,Y 205.191,Z 606.492,A -85,B 0,C 180,E1 -21170.029,E2 -21170.029} C_VEL
LIN {X 0,Y 204.627,Z 608.447,A -85,B 0,C 180,E1 -21172.196,E2 -21172.196} C_VEL
LIN {X 0,Y 203.983,Z 611.268,A -85,B 0,C 180,E1 -21176.608,E2 -21176.608} C_VEL
LIN {X 0,Y 203.866,Z 612.559,A -85,B 0,C 180,E1 -21180.484,E2 -21180.484} C_VEL
LIN {X 0,Y 204.112,Z 612.705,A -85,B 0,C 180,E1 -21184.28,E2 -21184.28} C_VEL
LIN {X 0,Y 204.775,Z 611.803,A -85,B 0,C 180,E1 -21188.152,E2 -21188.152} C_VEL
LIN {X 0,Y 205.751,Z 610.286,A -85,B 0,C 180,E1 -21191.288,E2 -21191.288} C_VEL
LIN {X 0,Y 207.561,Z 607.17,A -85,B 0,C 180,E1 -21195.319,E2 -21195.319} C_VEL
LIN {X 0,Y 209.783,Z 603.225,A -85,B 0,C 180,E1 -21198.915,E2 -21198.915} C_VEL
LIN {X 0,Y 212.728,Z 598.113,A -85,B 0,C 180,E1 -21202.455,E2 -21202.455} C_VEL
LIN {X 0,Y 216.693,Z 591.107,A -85,B 0,C 180,E1 -21206.178,E2 -21206.178} C_VEL
LIN {X 0,Y 221.009,Z 583.316,A -85,B 0,C 180,E1 -21209.421,E2 -21209.421} C_VEL
LIN {X 0,Y 225.538,Z 574.759,A -85,B 0,C 180,E1 -21212.279,E2 -21212.279} C_VEL
LIN {X 0,Y 230.528,Z 564.556,A -85,B 0,C 180,E1 -21215.021,E2 -21215.021} C_VEL
LIN {X 0,Y 235.781,Z 552.864,A -85,B 0,C 180,E1 -21217.517,E2 -21217.517} C_VEL
LIN {X 0,Y 240.695,Z 540.639,A -85,B 0,C 180,E1 -21219.6,E2 -21219.6} C_VEL
LIN {X 0,Y 245.272,Z 527.656,A -85,B 0,C 180,E1 -21221.376,E2 -21221.376} C_VEL
LIN {X 0,Y 249.576,Z 513.263,A -85,B 0,C 180,E1 -21222.92,E2 -21222.92} C_VEL
LIN {X 0,Y 253.081,Z 498.746,A -85,B 0,C 180,E1 -21224.127,E2 -21224.127} C_VEL
LIN {X 0,Y 255.926,Z 483.827,A -85,B 0,C 180,E1 -21225.038,E2 -21225.038} C_VEL
LIN {X 0,Y 257.998,Z 468.806,A -85,B 0,C 180,E1 -21225.672,E2 -21225.672} C_VEL
LIN {X 0,Y 264.302,Z 389.19,A -85,B 0,C 180,E1 -21227.885,E2 -21227.885} C_VEL
LIN {X 0,Y 260.058,Z 379.758,A -85,B 0,C 180,E1 -21229.842,E2 -21229.842} C_VEL
LIN {X 0,Y 257.061,Z 374.053,A -85,B 0,C 180,E1 -21231.287,E2 -21231.287} C_VEL
LIN {X 0,Y 253.157,Z 367.646,A -85,B 0,C 180,E1 -21233.31,E2 -21233.31} C_VEL
LIN {X 0,Y 248.406,Z 360.254,A -85,B 0,C 180,E1 -21236.121,E2 -21236.121} C_VEL
LIN {X 0,Y 246.082,Z 356.894,A -85,B 0,C 180,E1 -21237.674,E2 -21237.674} C_VEL
LIN {X 0,Y 243.253,Z 352.783,A -85,B 0,C 180,E1 -21239.838,E2 -21239.838} C_VEL
LIN {X 0,Y 240.235,Z 348.169,A -85,B 0,C 180,E1 -21242.675,E2 -21242.675} C_VEL
LIN {X 0,Y 237.139,Z 345.27,A -85,B 0,C 180,E1 -21246.288,E2 -21246.288} C_VEL
LIN {X 0,Y 236.052,Z 342.727,A -85,B 0,C 180,E1 -21248.348,E2 -21248.348} C_VEL
LIN {X 0,Y 234.305,Z 341.967,A -85,B 0,C 180,E1 -21253.887,E2 -21253.887} C_VEL
LIN {X 0,Y 235.194,Z 342.576,A -85,B 0,C 180,E1 -21259.556,E2 -21259.556} C_VEL
LIN {X 0,Y 235.485,Z 343.663,A -85,B 0,C 180,E1 -21260.473,E2 -21260.473} C_VEL
LIN {X 0,Y 235.633,Z 345.873,A -85,B 0,C 180,E1 -21261.291,E2 -21261.291} C_VEL
LIN {X 0,Y 236.027,Z 351.885,A -85,B 0,C 180,E1 -21263.103,E2 -21263.103} C_VEL
LIN {X 0,Y 236.534,Z 353.412,A -85,B 0,C 180,E1 -21264,E2 -21264} C_VEL
LIN {X 0,Y 238.165,Z 355.381,A -85,B 0,C 180,E1 -21266.019,E2 -21266.019} C_VEL
LIN {X 0,Y 239.267,Z 357.052,A -85,B 0,C 180,E1 -21267.21,E2 -21267.21} C_VEL
LIN {X 0,Y 242.635,Z 362.67,A -85,B 0,C 180,E1 -21270.333,E2 -21270.333} C_VEL
LIN {X 0,Y 245.317,Z 367.467,A -85,B 0,C 180,E1 -21272.411,E2 -21272.411} C_VEL
LIN {X 0,Y 249.007,Z 374.331,A -85,B 0,C 180,E1 -21274.878,E2 -21274.878} C_VEL
LIN {X 0,Y 253.179,Z 382.666,A -85,B 0,C 180,E1 -21277.314,E2 -21277.314} C_VEL
LIN {X 0,Y 257.61,Z 392.993,A -85,B 0,C 180,E1 -21279.667,E2 -21279.667} C_VEL
LIN {X 0,Y 259.778,Z 398.806,A -85,B 0,C 180,E1 -21280.757,E2 -21280.757} C_VEL
LIN {X 0,Y 253.212,Z 477.384,A -85,B 0,C 180,E1 -21282.944,E2 -21282.944} C_VEL
LIN {X 0,Y 250.851,Z 493.295,A -85,B 0,C 180,E1 -21283.612,E2 -21283.612} C_VEL
LIN {X 0,Y 247.578,Z 508.529,A -85,B 0,C 180,E1 -21284.504,E2 -21284.504} C_VEL
LIN {X 0,Y 243.721,Z 522.75,A -85,B 0,C 180,E1 -21285.633,E2 -21285.633} C_VEL
LIN {X 0,Y 239.052,Z 537.222,A -85,B 0,C 180,E1 -21287.169,E2 -21287.169} C_VEL
LIN {X 0,Y 234.077,Z 550.358,A -85,B 0,C 180,E1 -21288.947,E2 -21288.947} C_VEL
LIN {X 0,Y 228.968,Z 562.402,A -85,B 0,C 180,E1 -21291.009,E2 -21291.009} C_VEL
LIN {X 0,Y 223.723,Z 573.466,A -85,B 0,C 180,E1 -21293.356,E2 -21293.356} C_VEL
LIN {X 0,Y 218.123,Z 584.324,A -85,B 0,C 180,E1 -21296.236,E2 -21296.236} C_VEL
LIN {X 0,Y 212.86,Z 594.075,A -85,B 0,C 180,E1 -21299.546,E2 -21299.546} C_VEL
LIN {X 0,Y 208.408,Z 601.943,A -85,B 0,C 180,E1 -21302.92,E2 -21302.92} C_VEL
LIN {X 0,Y 204.451,Z 608.866,A -85,B 0,C 180,E1 -21306.716,E2 -21306.716} C_VEL
LIN {X 0,Y 201.534,Z 613.972,A -85,B 0,C 180,E1 -21310.321,E2 -21310.321} C_VEL
LIN {X 0,Y 199.694,Z 617.649,A -85,B 0,C 180,E1 -21313.648,E2 -21313.648} C_VEL
LIN {X 0,Y 198.109,Z 620.958,A -85,B 0,C 180,E1 -21317.712,E2 -21317.712} C_VEL
LIN {X 0,Y 197.347,Z 623.042,A -85,B 0,C 180,E1 -21321.811,E2 -21321.811} C_VEL
LIN {X 0,Y 197.169,Z 624.048,A -85,B 0,C 180,E1 -21326.457,E2 -21326.457} C_VEL
LIN {X 0,Y 197.401,Z 623.807,A -85,B 0,C 180,E1 -21330.001,E2 -21330.001} C_VEL
LIN {X 0,Y 197.253,Z 622.426,A -85,B 0,C 180,E1 -21334.087,E2 -21334.087} C_VEL
LIN {X 0,Y 197.388,Z 619.81,A -85,B 0,C 180,E1 -21338.189,E2 -21338.189} C_VEL
LIN {X 0,Y 198.048,Z 615.877,A -85,B 0,C 180,E1 -21342.294,E2 -21342.294} C_VEL
LIN {X 0,Y 199.435,Z 610.565,A -85,B 0,C 180,E1 -21346.375,E2 -21346.375} C_VEL
LIN {X 0,Y 201.64,Z 603.741,A -85,B 0,C 180,E1 -21350.399,E2 -21350.399} C_VEL
LIN {X 0,Y 204.601,Z 595.202,A -85,B 0,C 180,E1 -21354.343,E2 -21354.343} C_VEL
LIN {X 0,Y 207.609,Z 587.46,A -85,B 0,C 180,E1 -21357.194,E2 -21357.194} C_VEL
LIN {X 0,Y 210.795,Z 578.368,A -85,B 0,C 180,E1 -21360.007,E2 -21360.007} C_VEL
LIN {X 0,Y 214.561,Z 567.641,A -85,B 0,C 180,E1 -21362.715,E2 -21362.715} C_VEL
LIN {X 0,Y 218.473,Z 555.962,A -85,B 0,C 180,E1 -21365.101,E2 -21365.101} C_VEL
LIN {X 0,Y 222.339,Z 543.237,A -85,B 0,C 180,E1 -21367.195,E2 -21367.195} C_VEL
LIN {X 0,Y 225.936,Z 529.846,A -85,B 0,C 180,E1 -21368.951,E2 -21368.951} C_VEL
LIN {X 0,Y 229.135,Z 515.898,A -85,B 0,C 180,E1 -21370.386,E2 -21370.386} C_VEL
LIN {X 0,Y 231.951,Z 501.316,A -85,B 0,C 180,E1 -21371.514,E2 -21371.514} C_VEL
LIN {X 0,Y 234.192,Z 485.401,A -85,B 0,C 180,E1 -21372.398,E2 -21372.398} C_VEL
LIN {X 0,Y 235.546,Z 469.928,A -85,B 0,C 180,E1 -21372.968,E2 -21372.968} C_VEL
LIN {X 0,Y 240.594,Z 389.073,A -85,B 0,C 180,E1 -21375.338,E2 -21375.338} C_VEL
LIN {X 0,Y 233.736,Z 372.622,A -85,B 0,C 180,E1 -21377.438,E2 -21377.438} C_VEL
LIN {X 0,Y 224.96,Z 354.425,A -85,B 0,C 180,E1 -21380.274,E2 -21380.274} C_VEL
LIN {X 0,Y 217.499,Z 340.696,A -85,B 0,C 180,E1 -21382.851,E2 -21382.851} C_VEL
LIN {X 0,Y 211.011,Z 329.837,A -85,B 0,C 180,E1 -21385.261,E2 -21385.261} C_VEL
LIN {X 0,Y 208.924,Z 326.837,A -85,B 0,C 180,E1 -21386.066,E2 -21386.066} C_VEL
LIN {X 0,Y 206.162,Z 322.958,A -85,B 0,C 180,E1 -21387.161,E2 -21387.161} C_VEL
LIN {X 0,Y 203.65,Z 319.733,A -85,B 0,C 180,E1 -21388.172,E2 -21388.172} C_VEL
LIN {X 0,Y 202.813,Z 318.295,A -85,B 0,C 180,E1 -21388.538,E2 -21388.538} C_VEL
LIN {X 0,Y 200.678,Z 316.134,A -85,B 0,C 180,E1 -21389.406,E2 -21389.406} C_VEL
LIN {X 0,Y 199.711,Z 313.735,A -85,B 0,C 180,E1 -21389.9,E2 -21389.9} C_VEL
LIN {X 0,Y 199.624,Z 313.239,A -85,B 0,C 180,E1 -21390.031,E2 -21390.031} C_VEL
LIN {X 0,Y 199.624,Z 313.239,A -85,B 0,C 180,E1 -21392.759,E2 -21392.759} C_VEL
LIN {X 0,Y 199.662,Z 313.239,A -85,B 0,C 180,E1 -21397.217,E2 -21397.217} C_VEL
LIN {X 0,Y 199.748,Z 313.23,A -85,B 0,C 180,E1 -21401.8,E2 -21401.8} C_VEL
LIN {X 0,Y 199.801,Z 313.182,A -85,B 0,C 180,E1 -21405.743,E2 -21405.743} C_VEL
LIN {X 0,Y 200.024,Z 313.168,A -85,B 0,C 180,E1 -21409.879,E2 -21409.879} C_VEL
LIN {X 0,Y 199.99,Z 313.181,A -85,B 0,C 180,E1 -21413.945,E2 -21413.945} C_VEL
LIN {X 0,Y 200.258,Z 313.122,A -85,B 0,C 180,E1 -21417.986,E2 -21417.986} C_VEL
LIN {X 0,Y 200.44,Z 313.13,A -85,B 0,C 180,E1 -21419.997,E2 -21419.997} C_VEL
LIN {X 0,Y 199.979,Z 313.172,A -85,B 0,C 180,E1 -21424.027,E2 -21424.027} C_VEL
LIN {X 0,Y 200.053,Z 313.145,A -85,B 0,C 180,E1 -21428.075,E2 -21428.075} C_VEL
LIN {X 0,Y 199.861,Z 313.214,A -85,B 0,C 180,E1 -21432.177,E2 -21432.177} C_VEL
LIN {X 0,Y 199.758,Z 313.175,A -85,B 0,C 180,E1 -21436.344,E2 -21436.344} C_VEL
LIN {X 0,Y 199.649,Z 313.231,A -85,B 0,C 180,E1 -21440.607,E2 -21440.607} C_VEL
LIN {X 0,Y 199.612,Z 313.212,A -85,B 0,C 180,E1 -21444.988,E2 -21444.988} C_VEL
LIN {X 0,Y 199.596,Z 313.219,A -85,B 0,C 180,E1 -21449.531,E2 -21449.531} C_VEL
LIN {X 0,Y 199.656,Z 313.24,A -85,B 0,C 180,E1 -21452.349,E2 -21452.349} C_VEL
LIN {X 0,Y 199.607,Z 313.201,A -85,B 0,C 180,E1 -21456.762,E2 -21456.762} C_VEL
LIN {X 0,Y 199.584,Z 313.23,A -85,B 0,C 180,E1 -21459.329,E2 -21459.329} C_VEL
LIN {X 0,Y 199.556,Z 313.248,A -85,B 0,C 180,E1 -21462.304,E2 -21462.304} C_VEL
LIN {X 0,Y 199.566,Z 313.216,A -85,B 0,C 180,E1 -21465.225,E2 -21465.225} C_VEL
LIN {X 0,Y 199.566,Z 313.242,A -85,B 0,C 180,E1 -21468.002,E2 -21468.002} C_VEL
LIN {X 0,Y 199.595,Z 313.238,A -85,B 0,C 180,E1 -21470.766,E2 -21470.766} C_VEL
LIN {X 0,Y 199.6,Z 313.245,A -85,B 0,C 180,E1 -21475.711,E2 -21475.711} C_VEL
LIN {X 0,Y 199.68,Z 313.22,A -85,B 0,C 180,E1 -21478.133,E2 -21478.133} C_VEL
LIN {X 0,Y 199.628,Z 313.223,A -85,B 0,C 180,E1 -21480.553,E2 -21480.553} C_VEL
LIN {X 0,Y 200.487,Z 315.796,A -85,B 0,C 180,E1 -21481.027,E2 -21481.027} C_VEL
LIN {X 0,Y 202.548,Z 318.058,A -85,B 0,C 180,E1 -21481.881,E2 -21481.881} C_VEL
LIN {X 0,Y 203.314,Z 318.872,A -85,B 0,C 180,E1 -21482.188,E2 -21482.188} C_VEL
LIN {X 0,Y 205.422,Z 322.19,A -85,B 0,C 180,E1 -21483.081,E2 -21483.081} C_VEL
LIN {X 0,Y 206.838,Z 323.745,A -85,B 0,C 180,E1 -21483.631,E2 -21483.631} C_VEL
LIN {X 0,Y 209.612,Z 327.568,A -85,B 0,C 180,E1 -21484.713,E2 -21484.713} C_VEL
LIN {X 0,Y 216.624,Z 337.854,A -85,B 0,C 180,E1 -21487.283,E2 -21487.283} C_VEL
LIN {X 0,Y 223.378,Z 348.112,A -85,B 0,C 180,E1 -21489.56,E2 -21489.56} C_VEL
LIN {X 0,Y 233.33,Z 364.877,A -85,B 0,C 180,E1 -21492.65,E2 -21492.65} C_VEL
LIN {X 0,Y 236.788,Z 371.499,A -85,B 0,C 180,E1 -21493.673,E2 -21493.673} C_VEL
LIN {X 0,Y 240.882,Z 380.641,A -85,B 0,C 180,E1 -21494.881,E2 -21494.881} C_VEL
LIN {X 0,Y 235.29,Z 467.397,A -85,B 0,C 180,E1 -21497.438,E2 -21497.438} C_VEL
LIN {X 0,Y 233.407,Z 483.703,A -85,B 0,C 180,E1 -21498.218,E2 -21498.218} C_VEL
LIN {X 0,Y 231.103,Z 498.54,A -85,B 0,C 180,E1 -21499.265,E2 -21499.265} C_VEL
LIN {X 0,Y 228.317,Z 512.379,A -85,B 0,C 180,E1 -21500.551,E2 -21500.551} C_VEL
LIN {X 0,Y 224.754,Z 527.323,A -85,B 0,C 180,E1 -21502.362,E2 -21502.362} C_VEL
LIN {X 0,Y 221.128,Z 540.081,A -85,B 0,C 180,E1 -21504.299,E2 -21504.299} C_VEL
LIN {X 0,Y 217.067,Z 552.937,A -85,B 0,C 180,E1 -21506.751,E2 -21506.751} C_VEL
LIN {X 0,Y 213.04,Z 564.609,A -85,B 0,C 180,E1 -21509.527,E2 -21509.527} C_VEL
LIN {X 0,Y 209.513,Z 574.422,A -85,B 0,C 180,E1 -21512.402,E2 -21512.402} C_VEL
LIN {X 0,Y 205.896,Z 583.987,A -85,B 0,C 180,E1 -21515.877,E2 -21515.877} C_VEL
LIN {X 0,Y 202.935,Z 591.899,A -85,B 0,C 180,E1 -21519.467,E2 -21519.467} C_VEL
LIN {X 0,Y 200.679,Z 598.362,A -85,B 0,C 180,E1 -21523.156,E2 -21523.156} C_VEL
LIN {X 0,Y 198.865,Z 604.129,A -85,B 0,C 180,E1 -21527.424,E2 -21527.424} C_VEL
LIN {X 0,Y 197.868,Z 607.539,A -85,B 0,C 180,E1 -21530.804,E2 -21530.804} C_VEL
LIN {X 0,Y 197.001,Z 610.792,A -85,B 0,C 180,E1 -21535.345,E2 -21535.345} C_VEL
LIN {X 0,Y 196.795,Z 611.876,A -85,B 0,C 180,E1 -21537.661,E2 -21537.661} C_VEL
LIN {X 0,Y 196.771,Z 612.81,A -85,B 0,C 180,E1 -21541.005,E2 -21541.005} C_VEL
LIN {X 0,Y 197.092,Z 612.899,A -85,B 0,C 180,E1 -21544.908,E2 -21544.908} C_VEL
LIN {X 0,Y 198.099,Z 611.632,A -85,B 0,C 180,E1 -21549.685,E2 -21549.685} C_VEL
LIN {X 0,Y 198.959,Z 610.362,A -85,B 0,C 180,E1 -21552.154,E2 -21552.154} C_VEL
LIN {X 0,Y 200.502,Z 607.876,A -85,B 0,C 180,E1 -21555.495,E2 -21555.495} C_VEL
LIN {X 0,Y 203.084,Z 603.672,A -85,B 0,C 180,E1 -21559.58,E2 -21559.58} C_VEL
LIN {X 0,Y 206.188,Z 598.637,A -85,B 0,C 180,E1 -21563.223,E2 -21563.223} C_VEL
LIN {X 0,Y 210.034,Z 592.315,A -85,B 0,C 180,E1 -21566.772,E2 -21566.772} C_VEL
LIN {X 0,Y 214.799,Z 584.225,A -85,B 0,C 180,E1 -21570.295,E2 -21570.295} C_VEL
LIN {X 0,Y 219.964,Z 574.965,A -85,B 0,C 180,E1 -21573.455,E2 -21573.455} C_VEL
LIN {X 0,Y 225.204,Z 564.745,A -85,B 0,C 180,E1 -21576.237,E2 -21576.237} C_VEL
LIN {X 0,Y 230.094,Z 554.392,A -85,B 0,C 180,E1 -21578.502,E2 -21578.502} C_VEL
LIN {X 0,Y 235.343,Z 542.113,A -85,B 0,C 180,E1 -21580.662,E2 -21580.662} C_VEL
LIN {X 0,Y 240.334,Z 528.624,A -85,B 0,C 180,E1 -21582.555,E2 -21582.555} C_VEL
LIN {X 0,Y 244.788,Z 514.445,A -85,B 0,C 180,E1 -21584.106,E2 -21584.106} C_VEL
LIN {X 0,Y 248.608,Z 499.35,A -85,B 0,C 180,E1 -21585.377,E2 -21585.377} C_VEL
LIN {X 0,Y 251.604,Z 484.193,A -85,B 0,C 180,E1 -21586.308,E2 -21586.308} C_VEL
LIN {X 0,Y 253.832,Z 468.566,A -85,B 0,C 180,E1 -21586.963,E2 -21586.963} C_VEL
LIN {X 0,Y 260.157,Z 392.201,A -85,B 0,C 180,E1 -21589.102,E2 -21589.102} C_VEL
LIN {X 0,Y 255.504,Z 381.829,A -85,B 0,C 180,E1 -21591.417,E2 -21591.417} C_VEL
LIN {X 0,Y 251.063,Z 374.176,A -85,B 0,C 180,E1 -21593.788,E2 -21593.788} C_VEL
LIN {X 0,Y 246.457,Z 366.696,A -85,B 0,C 180,E1 -21596.642,E2 -21596.642} C_VEL
LIN {X 0,Y 244.298,Z 363.442,A -85,B 0,C 180,E1 -21598.165,E2 -21598.165} C_VEL
LIN {X 0,Y 241.531,Z 359.314,A -85,B 0,C 180,E1 -21600.377,E2 -21600.377} C_VEL
LIN {X 0,Y 238.499,Z 354.716,A -85,B 0,C 180,E1 -21603.381,E2 -21603.381} C_VEL
LIN {X 0,Y 235.906,Z 352.117,A -85,B 0,C 180,E1 -21606.632,E2 -21606.632} C_VEL
LIN {X 0,Y 234.932,Z 349.697,A -85,B 0,C 180,E1 -21608.605,E2 -21608.605} C_VEL
LIN {X 0,Y 233.332,Z 349,A -85,B 0,C 180,E1 -21615.731,E2 -21615.731} C_VEL
LIN {X 0,Y 234.816,Z 350.044,A -85,B 0,C 180,E1 -21620.898,E2 -21620.898} C_VEL
LIN {X 0,Y 236.534,Z 353.412,A -85,B 0,C 180,E1 -21624,E2 -21624} C_VEL
LIN {X 0,Y 237.079,Z 355,A -85,B 0,C 180,E1 -21624.867,E2 -21624.867} C_VEL
LIN {X 0,Y 237.618,Z 359.58,A -85,B 0,C 180,E1 -21626.062,E2 -21626.062} C_VEL
LIN {X 0,Y 238.264,Z 364.297,A -85,B 0,C 180,E1 -21627.242,E2 -21627.242} C_VEL
LIN {X 0,Y 239.023,Z 366.084,A -85,B 0,C 180,E1 -21628.082,E2 -21628.082} C_VEL
LIN {X 0,Y 240.878,Z 369.159,A -85,B 0,C 180,E1 -21629.791,E2 -21629.791} C_VEL
LIN {X 0,Y 243.352,Z 373.844,A -85,B 0,C 180,E1 -21631.818,E2 -21631.818} C_VEL
LIN {X 0,Y 247.24,Z 381.33,A -85,B 0,C 180,E1 -21634.529,E2 -21634.529} C_VEL
LIN {X 0,Y 251.457,Z 390.636,A -85,B 0,C 180,E1 -21637.114,E2 -21637.114} C_VEL
LIN {X 0,Y 255.1,Z 399.715,A -85,B 0,C 180,E1 -21639.145,E2 -21639.145} C_VEL
LIN {X 0,Y 255.741,Z 401.456,A -85,B 0,C 180,E1 -21639.482,E2 -21639.482} C_VEL
LIN {X 0,Y 249.142,Z 477.722,A -85,B 0,C 180,E1 -21641.625,E2 -21641.625} C_VEL
LIN {X 0,Y 246.693,Z 493.377,A -85,B 0,C 180,E1 -21642.286,E2 -21642.286} C_VEL
LIN {X 0,Y 243.324,Z 508.477,A -85,B 0,C 180,E1 -21643.174,E2 -21643.174} C_VEL
LIN {X 0,Y 239.332,Z 522.616,A -85,B 0,C 180,E1 -21644.296,E2 -21644.296} C_VEL
LIN {X 0,Y 234.502,Z 537.025,A -85,B 0,C 180,E1 -21645.831,E2 -21645.831} C_VEL
LIN {X 0,Y 229.334,Z 550.163,A -85,B 0,C 180,E1 -21647.61,E2 -21647.61} C_VEL
LIN {X 0,Y 224.49,Z 561.18,A -85,B 0,C 180,E1 -21649.49,E2 -21649.49} C_VEL
LIN {X 0,Y 218.969,Z 572.385,A -85,B 0,C 180,E1 -21651.843,E2 -21651.843} C_VEL
LIN {X 0,Y 213.851,Z 581.88,A -85,B 0,C 180,E1 -21654.316,E2 -21654.316} C_VEL
LIN {X 0,Y 208.43,Z 591.495,A -85,B 0,C 180,E1 -21657.459,E2 -21657.459} C_VEL
LIN {X 0,Y 203.356,Z 600.174,A -85,B 0,C 180,E1 -21661.065,E2 -21661.065} C_VEL
LIN {X 0,Y 199.858,Z 605.782,A -85,B 0,C 180,E1 -21663.926,E2 -21663.926} C_VEL
LIN {X 0,Y 196.117,Z 611.896,A -85,B 0,C 180,E1 -21667.898,E2 -21667.898} C_VEL
LIN {X 0,Y 193.366,Z 616.639,A -85,B 0,C 180,E1 -21672.006,E2 -21672.006} C_VEL
LIN {X 0,Y 191.877,Z 619.401,A -85,B 0,C 180,E1 -21675.145,E2 -21675.145} C_VEL
LIN {X 0,Y 190.634,Z 622.054,A -85,B 0,C 180,E1 -21679.379,E2 -21679.379} C_VEL
LIN {X 0,Y 190.116,Z 623.502,A -85,B 0,C 180,E1 -21683.634,E2 -21683.634} C_VEL
LIN {X 0,Y 190.154,Z 623.823,A -85,B 0,C 180,E1 -21687.883,E2 -21687.883} C_VEL
LIN {X 0,Y 190.302,Z 623.554,A -85,B 0,C 180,E1 -21690.001,E2 -21690.001} C_VEL
LIN {X 0,Y 190.146,Z 622.111,A -85,B 0,C 180,E1 -21694.24,E2 -21694.24} C_VEL
LIN {X 0,Y 190.326,Z 619.446,A -85,B 0,C 180,E1 -21698.495,E2 -21698.495} C_VEL
LIN {X 0,Y 191.051,Z 615.462,A -85,B 0,C 180,E1 -21702.752,E2 -21702.752} C_VEL
LIN {X 0,Y 192.553,Z 610.078,A -85,B 0,C 180,E1 -21706.978,E2 -21706.978} C_VEL
LIN {X 0,Y 194.914,Z 603.172,A -85,B 0,C 180,E1 -21711.136,E2 -21711.136} C_VEL
LIN {X 0,Y 197.608,Z 595.683,A -85,B 0,C 180,E1 -21714.702,E2 -21714.702} C_VEL
LIN {X 0,Y 201.193,Z 586.694,A -85,B 0,C 180,E1 -21718.137,E2 -21718.137} C_VEL
LIN {X 0,Y 204.587,Z 577.485,A -85,B 0,C 180,E1 -21721.016,E2 -21721.016} C_VEL
LIN {X 0,Y 208.528,Z 566.614,A -85,B 0,C 180,E1 -21723.787,E2 -21723.787} C_VEL
LIN {X 0,Y 212.63,Z 554.766,A -85,B 0,C 180,E1 -21726.215,E2 -21726.215} C_VEL
LIN {X 0,Y 216.628,Z 541.815,A -85,B 0,C 180,E1 -21728.35,E2 -21728.35} C_VEL
LIN {X 0,Y 219.96,Z 529.891,A -85,B 0,C 180,E1 -21729.926,E2 -21729.926} C_VEL
LIN {X 0,Y 223.451,Z 514.902,A -85,B 0,C 180,E1 -21731.488,E2 -21731.488} C_VEL
LIN {X 0,Y 226.406,Z 500.084,A -85,B 0,C 180,E1 -21732.617,E2 -21732.617} C_VEL
LIN {X 0,Y 228.578,Z 484.785,A -85,B 0,C 180,E1 -21733.468,E2 -21733.468} C_VEL
LIN {X 0,Y 230.047,Z 467.403,A -85,B 0,C 180,E1 -21734.104,E2 -21734.104} C_VEL
LIN {X 0,Y 234.971,Z 390.975,A -85,B 0,C 180,E1 -21736.383,E2 -21736.383} C_VEL
LIN {X 0,Y 228.252,Z 374.894,A -85,B 0,C 180,E1 -21738.546,E2 -21738.546} C_VEL
LIN {X 0,Y 220.274,Z 358.345,A -85,B 0,C 180,E1 -21741.241,E2 -21741.241} C_VEL
LIN {X 0,Y 213.223,Z 345.212,A -85,B 0,C 180,E1 -21743.793,E2 -21743.793} C_VEL
LIN {X 0,Y 207.203,Z 334.857,A -85,B 0,C 180,E1 -21746.148,E2 -21746.148} C_VEL
LIN {X 0,Y 202.63,Z 328.484,A -85,B 0,C 180,E1 -21747.993,E2 -21747.993} C_VEL
LIN {X 0,Y 199.827,Z 324.527,A -85,B 0,C 180,E1 -21749.188,E2 -21749.188} C_VEL
LIN {X 0,Y 197.03,Z 321.143,A -85,B 0,C 180,E1 -21750.412,E2 -21750.412} C_VEL
LIN {X 0,Y 196.063,Z 319.388,A -85,B 0,C 180,E1 -21750.889,E2 -21750.889} C_VEL
LIN {X 0,Y 193.751,Z 317.201,A -85,B 0,C 180,E1 -21751.935,E2 -21751.935} C_VEL
LIN {X 0,Y 192.72,Z 314.881,A -85,B 0,C 180,E1 -21752.51,E2 -21752.51} C_VEL
LIN {X 0,Y 192.596,Z 314.115,A -85,B 0,C 180,E1 -21752.712,E2 -21752.712} C_VEL
LIN {X 0,Y 192.648,Z 314.11,A -85,B 0,C 180,E1 -21756.338,E2 -21756.338} C_VEL
LIN {X 0,Y 192.696,Z 314.106,A -85,B 0,C 180,E1 -21761.489,E2 -21761.489} C_VEL
LIN {X 0,Y 192.727,Z 314.069,A -85,B 0,C 180,E1 -21765.208,E2 -21765.208} C_VEL
LIN {X 0,Y 192.946,Z 314.043,A -85,B 0,C 180,E1 -21769.564,E2 -21769.564} C_VEL
LIN {X 0,Y 192.955,Z 314.06,A -85,B 0,C 180,E1 -21773.723,E2 -21773.723} C_VEL
LIN {X 0,Y 193.204,Z 313.999,A -85,B 0,C 180,E1 -21777.912,E2 -21777.912} C_VEL
LIN {X 0,Y 193.406,Z 314.006,A -85,B 0,C 180,E1 -21779.997,E2 -21779.997} C_VEL
LIN {X 0,Y 192.926,Z 314.046,A -85,B 0,C 180,E1 -21784.175,E2 -21784.175} C_VEL
LIN {X 0,Y 193.007,Z 314.025,A -85,B 0,C 180,E1 -21788.371,E2 -21788.371} C_VEL
LIN {X 0,Y 192.787,Z 314.093,A -85,B 0,C 180,E1 -21792.631,E2 -21792.631} C_VEL
LIN {X 0,Y 192.712,Z 314.05,A -85,B 0,C 180,E1 -21796.959,E2 -21796.959} C_VEL
LIN {X 0,Y 192.579,Z 314.119,A -85,B 0,C 180,E1 -21801.4,E2 -21801.4} C_VEL
LIN {X 0,Y 192.612,Z 314.096,A -85,B 0,C 180,E1 -21804.19,E2 -21804.19} C_VEL
LIN {X 0,Y 192.587,Z 314.08,A -85,B 0,C 180,E1 -21808.858,E2 -21808.858} C_VEL
LIN {X 0,Y 192.586,Z 314.115,A -85,B 0,C 180,E1 -21813.183,E2 -21813.183} C_VEL
LIN {X 0,Y 192.532,Z 314.092,A -85,B 0,C 180,E1 -21818.351,E2 -21818.351} C_VEL
LIN {X 0,Y 192.474,Z 314.117,A -85,B 0,C 180,E1 -21823.09,E2 -21823.09} C_VEL
LIN {X 0,Y 192.477,Z 314.107,A -85,B 0,C 180,E1 -21826.903,E2 -21826.903} C_VEL
LIN {X 0,Y 192.537,Z 314.105,A -85,B 0,C 180,E1 -21831.645,E2 -21831.645} C_VEL
LIN {X 0,Y 192.585,Z 314.122,A -85,B 0,C 180,E1 -21836.811,E2 -21836.811} C_VEL
LIN {X 0,Y 192.631,Z 314.1,A -85,B 0,C 180,E1 -21837.904,E2 -21837.904} C_VEL
LIN {X 0,Y 193.581,Z 316.891,A -85,B 0,C 180,E1 -21838.498,E2 -21838.498} C_VEL
LIN {X 0,Y 195.482,Z 318.985,A -85,B 0,C 180,E1 -21839.382,E2 -21839.382} C_VEL
LIN {X 0,Y 196.427,Z 319.888,A -85,B 0,C 180,E1 -21839.8,E2 -21839.8} C_VEL
LIN {X 0,Y 198.486,Z 323.114,A -85,B 0,C 180,E1 -21840.767,E2 -21840.767} C_VEL
LIN {X 0,Y 200.169,Z 325.013,A -85,B 0,C 180,E1 -21841.483,E2 -21841.483} C_VEL
LIN {X 0,Y 202.772,Z 328.571,A -85,B 0,C 180,E1 -21842.584,E2 -21842.584} C_VEL
LIN {X 0,Y 207.76,Z 335.68,A -85,B 0,C 180,E1 -21844.599,E2 -21844.599} C_VEL
LIN {X 0,Y 215.008,Z 346.254,A -85,B 0,C 180,E1 -21847.274,E2 -21847.274} C_VEL
LIN {X 0,Y 222.023,Z 357.598,A -85,B 0,C 180,E1 -21849.684,E2 -21849.684} C_VEL
LIN {X 0,Y 231.352,Z 373.941,A -85,B 0,C 180,E1 -21852.621,E2 -21852.621} C_VEL
LIN {X 0,Y 235.256,Z 382.865,A -85,B 0,C 180,E1 -21853.844,E2 -21853.844} C_VEL
LIN {X 0,Y 229.615,Z 467.719,A -85,B 0,C 180,E1 -21856.39,E2 -21856.39} C_VEL
LIN {X 0,Y 227.691,Z 483.937,A -85,B 0,C 180,E1 -21857.182,E2 -21857.182} C_VEL
LIN {X 0,Y 225.211,Z 499.331,A -85,B 0,C 180,E1 -21858.296,E2 -21858.296} C_VEL
LIN {X 0,Y 222.458,Z 512.446,A -85,B 0,C 180,E1 -21859.533,E2 -21859.533} C_VEL
LIN {X 0,Y 219.047,Z 526.403,A -85,B 0,C 180,E1 -21861.233,E2 -21861.233} C_VEL
LIN {X 0,Y 215.31,Z 539.312,A -85,B 0,C 180,E1 -21863.204,E2 -21863.204} C_VEL
LIN {X 0,Y 211.068,Z 552.298,A -85,B 0,C 180,E1 -21865.681,E2 -21865.681} C_VEL
LIN {X 0,Y 206.837,Z 564.199,A -85,B 0,C 180,E1 -21868.539,E2 -21868.539} C_VEL
LIN {X 0,Y 203.329,Z 573.626,A -85,B 0,C 180,E1 -21871.338,E2 -21871.338} C_VEL
LIN {X 0,Y 199.352,Z 583.769,A -85,B 0,C 180,E1 -21875.055,E2 -21875.055} C_VEL
LIN {X 0,Y 196.239,Z 591.751,A -85,B 0,C 180,E1 -21878.754,E2 -21878.754} C_VEL
LIN {X 0,Y 193.816,Z 598.271,A -85,B 0,C 180,E1 -21882.565,E2 -21882.565} C_VEL
LIN {X 0,Y 192.282,Z 602.818,A -85,B 0,C 180,E1 -21885.909,E2 -21885.909} C_VEL
LIN {X 0,Y 191.181,Z 606.554,A -85,B 0,C 180,E1 -21889.319,E2 -21889.319} C_VEL
LIN {X 0,Y 190.317,Z 609.269,A -85,B 0,C 180,E1 -21892.614,E2 -21892.614} C_VEL
LIN {X 0,Y 189.731,Z 611.873,A -85,B 0,C 180,E1 -21897.261,E2 -21897.261} C_VEL
LIN {X 0,Y 189.694,Z 613.046,A -85,B 0,C 180,E1 -21901.564,E2 -21901.564} C_VEL
LIN {X 0,Y 190.175,Z 612.988,A -85,B 0,C 180,E1 -21906.246,E2 -21906.246} C_VEL
LIN {X 0,Y 190.89,Z 612.163,A -85,B 0,C 180,E1 -21909.369,E2 -21909.369} C_VEL
LIN {X 0,Y 192.567,Z 609.863,A -85,B 0,C 180,E1 -21913.9,E2 -21913.9} C_VEL
LIN {X 0,Y 194.639,Z 606.815,A -85,B 0,C 180,E1 -21917.745,E2 -21917.745} C_VEL
LIN {X 0,Y 197.438,Z 602.641,A -85,B 0,C 180,E1 -21921.543,E2 -21921.543} C_VEL
LIN {X 0,Y 200.785,Z 597.475,A -85,B 0,C 180,E1 -21925.119,E2 -21925.119} C_VEL
LIN {X 0,Y 205.268,Z 590.498,A -85,B 0,C 180,E1 -21928.862,E2 -21928.862} C_VEL
LIN {X 0,Y 209.933,Z 582.912,A -85,B 0,C 180,E1 -21932.055,E2 -21932.055} C_VEL
LIN {X 0,Y 215.257,Z 573.812,A -85,B 0,C 180,E1 -21935.106,E2 -21935.106} C_VEL
LIN {X 0,Y 220.894,Z 563.281,A -85,B 0,C 180,E1 -21937.913,E2 -21937.913} C_VEL
LIN {X 0,Y 226.072,Z 552.636,A -85,B 0,C 180,E1 -21940.187,E2 -21940.187} C_VEL
LIN {X 0,Y 231.487,Z 540.094,A -85,B 0,C 180,E1 -21942.329,E2 -21942.329} C_VEL
LIN {X 0,Y 236.211,Z 527.708,A -85,B 0,C 180,E1 -21944.009,E2 -21944.009} C_VEL
LIN {X 0,Y 240.495,Z 514.409,A -85,B 0,C 180,E1 -21945.462,E2 -21945.462} C_VEL
LIN {X 0,Y 244.374,Z 499.687,A -85,B 0,C 180,E1 -21946.702,E2 -21946.702} C_VEL
LIN {X 0,Y 247.534,Z 484.343,A -85,B 0,C 180,E1 -21947.643,E2 -21947.643} C_VEL
LIN {X 0,Y 249.756,Z 469.385,A -85,B 0,C 180,E1 -21948.274,E2 -21948.274} C_VEL
LIN {X 0,Y 256.082,Z 395.103,A -85,B 0,C 180,E1 -21950.385,E2 -21950.385} C_VEL
LIN {X 0,Y 252.186,Z 386.364,A -85,B 0,C 180,E1 -21952.481,E2 -21952.481} C_VEL
LIN {X 0,Y 248.327,Z 379.603,A -85,B 0,C 180,E1 -21954.688,E2 -21954.688} C_VEL
LIN {X 0,Y 244.36,Z 372.898,A -85,B 0,C 180,E1 -21957.292,E2 -21957.292} C_VEL
LIN {X 0,Y 242.417,Z 369.855,A -85,B 0,C 180,E1 -21958.752,E2 -21958.752} C_VEL
LIN {X 0,Y 239.122,Z 364.775,A -85,B 0,C 180,E1 -21961.614,E2 -21961.614} C_VEL
LIN {X 0,Y 237.237,Z 361.643,A -85,B 0,C 180,E1 -21963.632,E2 -21963.632} C_VEL
LIN {X 0,Y 234.614,Z 358.832,A -85,B 0,C 180,E1 -21967.101,E2 -21967.101} C_VEL
LIN {X 0,Y 233.755,Z 356.647,A -85,B 0,C 180,E1 -21968.995,E2 -21968.995} C_VEL
LIN {X 0,Y 232.362,Z 356.045,A -85,B 0,C 180,E1 -21975.799,E2 -21975.799} C_VEL
LIN {X 0,Y 233.671,Z 356.927,A -85,B 0,C 180,E1 -21980.545,E2 -21980.545} C_VEL
LIN {X 0,Y 235.569,Z 360.599,A -85,B 0,C 180,E1 -21984.058,E2 -21984.058} C_VEL
LIN {X 0,Y 237.126,Z 362.617,A -85,B 0,C 180,E1 -21986.013,E2 -21986.013} C_VEL
LIN {X 0,Y 239.023,Z 366.084,A -85,B 0,C 180,E1 -21988.082,E2 -21988.082} C_VEL
LIN {X 0,Y 239.898,Z 367.541,A -85,B 0,C 180,E1 -21988.921,E2 -21988.921} C_VEL
LIN {X 0,Y 240.985,Z 370.938,A -85,B 0,C 180,E1 -21990.038,E2 -21990.038} C_VEL
LIN {X 0,Y 241.867,Z 375.144,A -85,B 0,C 180,E1 -21991.016,E2 -21991.016} C_VEL
LIN {X 0,Y 243.746,Z 384.178,A -85,B 0,C 180,E1 -21992.922,E2 -21992.922} C_VEL
LIN {X 0,Y 244.66,Z 386.769,A -85,B 0,C 180,E1 -21993.626,E2 -21993.626} C_VEL
LIN {X 0,Y 248.504,Z 395.644,A -85,B 0,C 180,E1 -21996.17,E2 -21996.17} C_VEL
LIN {X 0,Y 251.884,Z 404.441,A -85,B 0,C 180,E1 -21998.184,E2 -21998.184} C_VEL
LIN {X 0,Y 245.35,Z 476.989,A -85,B 0,C 180,E1 -22000.223,E2 -22000.223} C_VEL
LIN {X 0,Y 242.827,Z 492.812,A -85,B 0,C 180,E1 -22000.879,E2 -22000.879} C_VEL
LIN {X 0,Y 239.213,Z 508.537,A -85,B 0,C 180,E1 -22001.8,E2 -22001.8} C_VEL
LIN {X 0,Y 235.101,Z 522.618,A -85,B 0,C 180,E1 -22002.915,E2 -22002.915} C_VEL
LIN {X 0,Y 230.635,Z 535.556,A -85,B 0,C 180,E1 -22004.269,E2 -22004.269} C_VEL
LIN {X 0,Y 225.629,Z 547.976,A -85,B 0,C 180,E1 -22005.914,E2 -22005.914} C_VEL
LIN {X 0,Y 220.157,Z 559.961,A -85,B 0,C 180,E1 -22007.906,E2 -22007.906} C_VEL
LIN {X 0,Y 214.413,Z 571.308,A -85,B 0,C 180,E1 -22010.272,E2 -22010.272} C_VEL
LIN {X 0,Y 209.022,Z 580.948,A -85,B 0,C 180,E1 -22012.757,E2 -22012.757} C_VEL
LIN {X 0,Y 203.362,Z 590.456,A -85,B 0,C 180,E1 -22015.836,E2 -22015.836} C_VEL
LIN {X 0,Y 199.103,Z 597.399,A -85,B 0,C 180,E1 -22018.626,E2 -22018.626} C_VEL
LIN {X 0,Y 194.584,Z 604.198,A -85,B 0,C 180,E1 -22021.998,E2 -22021.998} C_VEL
LIN {X 0,Y 190.426,Z 610.582,A -85,B 0,C 180,E1 -22026.049,E2 -22026.049} C_VEL
LIN {X 0,Y 187.202,Z 615.594,A -85,B 0,C 180,E1 -22030.254,E2 -22030.254} C_VEL
LIN {X 0,Y 184.955,Z 619.356,A -85,B 0,C 180,E1 -22034.576,E2 -22034.576} C_VEL
LIN {X 0,Y 183.597,Z 621.944,A -85,B 0,C 180,E1 -22038.967,E2 -22038.967} C_VEL
LIN {X 0,Y 183.035,Z 623.347,A -85,B 0,C 180,E1 -22043.386,E2 -22043.386} C_VEL
LIN {X 0,Y 183.048,Z 623.6,A -85,B 0,C 180,E1 -22047.801,E2 -22047.801} C_VEL
LIN {X 0,Y 183.204,Z 623.298,A -85,B 0,C 180,E1 -22050.001,E2 -22050.001} C_VEL
LIN {X 0,Y 183.044,Z 621.785,A -85,B 0,C 180,E1 -22054.405,E2 -22054.405} C_VEL
LIN {X 0,Y 183.261,Z 619.047,A -85,B 0,C 180,E1 -22058.825,E2 -22058.825} C_VEL
LIN {X 0,Y 184.066,Z 615.009,A -85,B 0,C 180,E1 -22063.244,E2 -22063.244} C_VEL
LIN {X 0,Y 185.694,Z 609.556,A -85,B 0,C 180,E1 -22067.625,E2 -22067.625} C_VEL
LIN {X 0,Y 188.216,Z 602.559,A -85,B 0,C 180,E1 -22071.926,E2 -22071.926} C_VEL
LIN {X 0,Y 191.106,Z 594.984,A -85,B 0,C 180,E1 -22075.602,E2 -22075.602} C_VEL
LIN {X 0,Y 194.327,Z 587.272,A -85,B 0,C 180,E1 -22078.633,E2 -22078.633} C_VEL
LIN {X 0,Y 197.86,Z 578.064,A -85,B 0,C 180,E1 -22081.65,E2 -22081.65} C_VEL
LIN {X 0,Y 201.846,Z 567.524,A -85,B 0,C 180,E1 -22084.458,E2 -22084.458} C_VEL
LIN {X 0,Y 206.04,Z 555.891,A -85,B 0,C 180,E1 -22086.955,E2 -22086.955} C_VEL
LIN {X 0,Y 210.187,Z 543.23,A -85,B 0,C 180,E1 -22089.133,E2 -22089.133} C_VEL
LIN {X 0,Y 214.169,Z 529.353,A -85,B 0,C 180,E1 -22091.018,E2 -22091.018} C_VEL
LIN {X 0,Y 217.634,Z 514.96,A -85,B 0,C 180,E1 -22092.542,E2 -22092.542} C_VEL
LIN {X 0,Y 220.684,Z 500.237,A -85,B 0,C 180,E1 -22093.683,E2 -22093.683} C_VEL
LIN {X 0,Y 222.919,Z 485.107,A -85,B 0,C 180,E1 -22094.546,E2 -22094.546} C_VEL
LIN {X 0,Y 224.338,Z 469.694,A -85,B 0,C 180,E1 -22095.136,E2 -22095.136} C_VEL
LIN {X 0,Y 229.502,Z 393.273,A -85,B 0,C 180,E1 -22097.438,E2 -22097.438} C_VEL
LIN {X 0,Y 223.414,Z 378.565,A -85,B 0,C 180,E1 -22099.502,E2 -22099.502} C_VEL
LIN {X 0,Y 215.957,Z 362.825,A -85,B 0,C 180,E1 -22102.136,E2 -22102.136} C_VEL
LIN {X 0,Y 209.191,Z 350.001,A -85,B 0,C 180,E1 -22104.704,E2 -22104.704} C_VEL
LIN {X 0,Y 203.481,Z 340.021,A -85,B 0,C 180,E1 -22107.035,E2 -22107.035} C_VEL
LIN {X 0,Y 198.648,Z 333.335,A -85,B 0,C 180,E1 -22109.059,E2 -22109.059} C_VEL
LIN {X 0,Y 195.61,Z 329.193,A -85,B 0,C 180,E1 -22110.423,E2 -22110.423} C_VEL
LIN {X 0,Y 192.539,Z 324.985,A -85,B 0,C 180,E1 -22111.891,E2 -22111.891} C_VEL
LIN {X 0,Y 190.141,Z 322.065,A -85,B 0,C 180,E1 -22113.074,E2 -22113.074} C_VEL
LIN {X 0,Y 189.296,Z 320.414,A -85,B 0,C 180,E1 -22113.54,E2 -22113.54} C_VEL
LIN {X 0,Y 186.919,Z 318.449,A -85,B 0,C 180,E1 -22114.701,E2 -22114.701} C_VEL
LIN {X 0,Y 185.753,Z 316.038,A -85,B 0,C 180,E1 -22115.402,E2 -22115.402} C_VEL
LIN {X 0,Y 185.573,Z 314.994,A -85,B 0,C 180,E1 -22115.609,E2 -22115.609} C_VEL
LIN {X 0,Y 185.627,Z 314.985,A -85,B 0,C 180,E1 -22121.176,E2 -22121.176} C_VEL
LIN {X 0,Y 185.71,Z 314.926,A -85,B 0,C 180,E1 -22126.872,E2 -22126.872} C_VEL
